// TwinCAT 3 PLC project Untitled1
// ProgramVersion: 3.1.4023.0
// libraries:
//   Tc2_ControllerToolbox, * (Beckhoff Automation GmbH)
//   Tc2_Standard, * (Beckhoff Automation GmbH)
//   Tc2_System, * (Beckhoff Automation GmbH)
//   Tc2_TempController, * (Beckhoff Automation GmbH)
//   Tc2_Utilities, * (Beckhoff Automation GmbH)
//   Tc3_EventLogger, * (Beckhoff Automation GmbH)
//   Tc3_Module, * (Beckhoff Automation GmbH)
// project tree:
//   DUTs/01_系统/ ST_AlarmID.TcDUT, ST_AlarmString.TcDUT, ST_Input.TcDUT, ST_Output.TcDUT, ST_Setting.TcDUT, ST_States.TcDUT
//   DUTs/Data types Alarm/ Alm_AlarmHistoryType.TcDUT, Alm_AlarmType.TcDUT, Alm_AlmMsg.TcDUT, Alm_EventClass.TcDUT
//   DUTs/ ST_Point.TcDUT
//   DUTs/文件配方/ FB_FileOperate.TcPOU
//   DUTs/文件配方/Swen_Products/ FB_DirectoryCopy.TcPOU, FB_FileCopy.TcPOU, FB_FileCopy_lib.TcPOU
//   GVLs/ Visu_Variables_HideInput.TcGVL, _01_Global_Variables.TcGVL, _04_Global_Variables_InOutput.TcGVL, _10_Global_Variables_Alarm.TcGVL, _12_Global_Variables_PeiFan.TcGVL
//   / PlcTask.TcTTO
//   POUs/ Controller_v2.TcPOU, FB_Actuator.TcPOU, Line_chart.TcPOU, MAIN.TcPOU
//   POUs/EventGridTest/ EventGrid.TcPOU
//   POUs/报警/ FB_AlarmMain.TcPOU, FB_SetAlarm.TcPOU, MAIN_Alarm.TcPOU, SW_FormatWstring.TcPOU
//   POUs/文件记录/ data_save.TcPOU, FB_DiagDataLogging.TcPOU
// real-time tasks:
//   TASK PlcTask: cycle T#10ms, priority 20, ADS port 350

CONFIGURATION Untitled1
    RESOURCE PLC ON TwinCAT3
        TASK PlcTask(INTERVAL := T#10ms, PRIORITY := 20);
        PROGRAM MAIN WITH PlcTask : MAIN;
    END_RESOURCE
END_CONFIGURATION

// ---- DUTs/01_系统/ST_AlarmID.TcDUT
TYPE ST_AlarmID :
(*报警的id号，swen*)
STRUCT
	(*系统*)
	EtherCATBusErr:					INT:=1;(*EtherCAT总线错误*)
	SystemLoading:					INT:=2;(*系统启动中*)
	EmergentStop:					INT:=3;(*急停按钮*)
	ProductChangeNeedSave:			INT:=4;
	ProductLoadingNoPowerOff:		INT:=5;
	AirPressLow:					INT:=6;(*气压低!*)
	Prushing:						INT:=7;(*暂停中*)
	NeedHoming:						INT:=8;(*开机前请先找原点*)
	IsHoming:						INT:=9;(*正在找原点*)
	AutoStoping:					INT:=10;(*自动停机中*)
	AutoStopImediery:				INT:=11;(*马上停机中*)
	AutoRuning:						INT:=12;(*设备运行中*)
	ComErrorVS:						INT:=13;(*视觉控制器通讯异常*)
	ServoError:						INT:=14;(*伺服出错*)
	ServoHwError:					INT:=15;(*伺服驱动器报错，硬件报错*)
	ServoLimit:						INT:=16;(*伺服驱动器限位到*)
	CycleTimeOut:					INT:=17;(*循环时间超时*)
	ModbusRtuError:					INT:=18;(*ModbusRtu总线错误*)
	RobotError1:					INT:=19;(*机器人错误*)
	RobotError2:					INT:=20;(*机器人错误*)
	StepServoError:					INT:=21;(*步进驱动器报错*)
	RobotSN_Error:					INT:=22;(*机器人序列号异常*)

	(*程序逻辑*)
	ClampVacuum:					INT:=26;(*机器人1真空吸取失败*)








	(*序列号*)
	Machime_SoftHwDif:				INT:=50;(*软硬件不匹配*)
	Machime_Alarm_NeedKey:			INT:=51;(*系统即将进入维护模式*)
	Machime_Stop_NeedKey:			INT:=52;(*系统已经进入维护模式*)

END_STRUCT
END_TYPE

// ---- DUTs/01_系统/ST_AlarmString.TcDUT
TYPE ST_AlarmString :
STRUCT
	chinese:		STRING:='CN';
	english:		STRING:='EN';
END_STRUCT
END_TYPE

// ---- DUTs/01_系统/ST_Input.TcDUT
TYPE ST_Input :
STRUCT
	biSnAirPressOk:				BOOL;(*压缩气源正常*)
	biSnBackDoorIsClose:				BOOL;(*后门关*)

	biSwEmgStop:				BOOL;(*急停按钮*)
	biBtStart:				BOOL;(*开始按钮*)
	biBtStop:				BOOL;(*停止按钮*)
	biBtHold:				BOOL;(*暂停按钮*)

   	biSnVacuuSor:				BOOL;(*取料真空检测*)

	biSnConvBoxIn:				BOOL;(*检测到进料口有箱子进来了*)
	biSnConvBoxOut:				BOOL;(*检测到出料口有箱子需要出来*)
	biSnBoxCapper:				BOOL;(*封箱机检测到有箱子进来*)


	noUse:				BOOL;





END_STRUCT
END_TYPE

// ---- DUTs/01_系统/ST_Output.TcDUT
TYPE ST_Output :
STRUCT


  	bqBoxCapperDw     (*	 压箱气缸	*)	,
  	bqBoxCapperCut      (*	剪断气缸  	*)	,

	bqClamperSuck	(*	机械手吸真空		*)	,
 	bqClamperZBrake          (*Z伺服刹车*)	,

	bqLightGrean(*绿灯 *)	,
 	bqLightYellow(*黄灯*)	,
 	bqLightRed(*红灯*)	,
 	bqBuzzer(*蜂鸣器*)	,

	noUse:				BOOL;

END_STRUCT
END_TYPE

// ---- DUTs/01_系统/ST_Setting.TcDUT
TYPE ST_Setting :
STRUCT
	(*系统*)
	gcSimulationMode:		BOOL;
	JogVelocity:			REAL:=20;
	AutoVelocity:			REAL:=500;(*皮带的速度*)
	ClampVelocity:			REAL:=2000;(*机械手的速度*)

	tCutTime:				REAL:=0.5;(*剪断时间*)

	ZPickUpHeight:			REAL:=200;(*抓起来的高度*)
	XPlacePos:				REAL:=450;(*抓过去的X距离*)
	YPlacePos:				REAL:=330;(*抓过去的Y距离*)
	ZPlacePos:				REAL:=-650;(*放到地板的高度*)
	Box_Longth:				REAL:=215;(*箱子长*)
	Box_Width:				REAL:=190;(*箱子宽*)
	Box_Height:				REAL:=198;(*箱子高*)

END_STRUCT
END_TYPE

// ---- DUTs/01_系统/ST_States.TcDUT
TYPE ST_States :
STRUCT
	ManualModeIsActive:				BOOL;(*手动模式*)
	AutoModeIsActive:				BOOL;(*自动模式*)
	MachineRunInCycle:				BOOL;(*自动运行中*)
	GoPauseState:					BOOL;(*请求暂停记忆*)
	AutoStoping:						BOOL;(*自动停机中*)
	ResetAlarm:						BOOL;(*报警复位*)
	GoHome:							BOOL;(*请求找原点*)


	(*电机*)
	HomeDone:						BOOL;(*原点完成*)
	Motor_PowerOn:				BOOL;(*上电完成*)
	Motor_HomeDone:				BOOL;(*原点完成*)
	Motor_SwError:				BOOL;(*电机NC软件出错*)
	Motor_SwErrId:				UDINT;
	Motor_Limit:				BOOL;(*电机限位*)
	Motor_HwError:				BOOL;(*电机硬件出错*)

	Hmi_btHome:						BOOL;(*画面按钮*)(*回原点*)
	Hmi_btAutoRun:					BOOL;(*画面按钮*)(*开始*)
	Hmi_btAutoStop:					BOOL;(*画面按钮*)(*停止*)
	Hmi_btPause:					BOOL;(*画面按钮*)(*暂停*)


	(*状态*)
	ConvCanRun:						BOOL:=TRUE;(*传送带启动允许*)

	ActBoxId:						INT;(*当前进箱子的ID号*)


END_STRUCT
END_TYPE

// ---- DUTs/Data types Alarm/Alm_AlarmHistoryType.TcDUT
TYPE Alm_AlarmHistoryType :
STRUCT
  	EventMessage:            	WSTRING;
	EventId:					INT;
   	EventTime:               	DT;
END_STRUCT
END_TYPE

// ---- DUTs/Data types Alarm/Alm_AlarmType.TcDUT
TYPE Alm_AlarmType :
STRUCT
      (*InPut*)
	EventId:					INT;
    EventMessage:			WSTRING;
    EventTime:                                 DT;
	EventActive:				BOOL;
	QuitRequired:				BOOL;
	QuitEvent:				BOOL;
	EventClass:				Alm_EventClass;
	AlarmMsg:				Alm_AlmMsg;
	AlarmlampOn:			BOOL;(*报警灯*)
	AutoRunOff:				BOOL;(*退出自动循环*)

	(* event actions OutPut	*)
	AlarmAction1:				BOOL;
	AlarmAction2:				BOOL;
	AlarmAction3:				BOOL;
	AlarmAction4:				BOOL;
	AlarmAction5:				BOOL;
	AlarmAction6:				BOOL;
	AlarmAction7:				BOOL;
	AlarmAction8:				BOOL;

       (*OutPut*)
	EventAlive:					BOOL;
    ShowlampOn:           		BOOL;
	InUse:                		BOOL;
END_STRUCT
END_TYPE;

// ---- DUTs/Data types Alarm/Alm_AlmMsg.TcDUT
TYPE Alm_AlmMsg :
STRUCT
	CN:		WSTRING:="中文";
	EN:		STRING:='En';	
END_STRUCT
END_TYPE

// ---- DUTs/Data types Alarm/Alm_EventClass.TcDUT
TYPE Alm_EventClass :
(
    NoAlarm                  :=0,(*无警报*)
    Message_1      :=1,(*信息*)
    Event_2            :=2,(*事件*)
    non_3                        :=3,(*暂无*)
    non_4                       :=4,(*暂无*)
    non_5                         :=5,(*暂无*)
    Alarm_6          :=6,(*不停机警报*)
    Stop_7                :=7(*停机警报*)
);
END_TYPE

// ---- DUTs/ST_Point.TcDUT
TYPE ST_Point :
STRUCT
	x : LREAL;
	y : LREAL;
END_STRUCT
END_TYPE

// ---- GVLs/Visu_Variables_HideInput.TcGVL
{attribute 'Tc2GvlVarNames'}
VAR_GLOBAL

	(*
		User Level Control
	*)
	sUserLevel:					STRING[20];
	nVisuUserLevel:				INT;
	bUseLogOutDelay:			BOOL;
	fUserLogOutDelay:			LREAL;
	sUserPassword:				STRING[20];
	bUserLevel0:				BOOL;
	bUserLevel1:				BOOL;
	bUserLevel2:				BOOL;
	bUserLevel3:				BOOL;
	bNewPassword:				BOOL;
	sNewUserPass1:			STRING[20];
	sNewUserPass2:			STRING[20];
	oldPasswords:				ARRAY [0..7] OF STRING[20];
	oldLanguage:				STRING[40];
	bVisuExUserLevel:			BOOL;
	bVisuInUserLevel:			BOOL;

(* ######################### Pswd Input Varaibles ########################## *)

	sPassInput : STRING := '';
	sPassV : STRING;

	i: DINT;
	iLen: DINT;
	bReset: BOOL;

	b_a_s : BOOL;
	b_b_s : BOOL;
	b_c_s : BOOL;
	b_d_s : BOOL;
	b_e_s : BOOL;
	b_f_s : BOOL;




	b_1_s : BOOL;
	b_2_s : BOOL;
	b_3_s : BOOL;
	b_4_s : BOOL;
	b_5_s : BOOL;
	b_6_s : BOOL;
	b_7_s : BOOL;
	b_8_s : BOOL;
	b_9_s : BOOL;
	b_0_s : BOOL;



	bBack: BOOL;
	iBackLen: INT;
	bShowNumPad:	BOOL;
	bHideNumPad:	BOOL;
	bCmdShowNumPad: BOOL;
	bCmdEnterValue:	BOOL;
	bCmdEscNumPad:	BOOL;
	sChangedPswd: STRING;

	bCmdShowNumPadUserPswd:	BOOL;
	bCmdShowNumPadNewPswd1:	BOOL;
	bCmdShowNumPadNewPswd2:	BOOL;

	sUserPasswordHide	:	STRING[20];
	sNewUserPass1Hide:	STRING[20];
	sNewUserPass2Hide:	STRING[20];

	bHidePswdFlush:	BOOL;

END_VAR

// ---- GVLs/_01_Global_Variables.TcGVL
{attribute 'Tc2GvlVarNames'}
VAR_GLOBAL
	DATA:						ST_States;	(*状态*)
//	gBox: 						ARRAY[0..23] OF ST_Box;(*箱子的状态*)
//	CLAMP:						APP_Clamp;(*实例化FB APP_Clmap*)
//	CONV:						APP_Conv;(*实例化FB APP_Conv*)

	RqSysManualModeIsActive,		(*需要在手动模式*)
	RqSysAutoModeIsActive,			(*需要在自动模式*)
	RqSysGoHome:				BOOL;(*需要回原点信号*)
	RqSysMachineRunInCycle: 	BOOL;(*需要设备在循环运行模式*)
	RqSysGoPauseState: 			BOOL;(*需要设备暂停*)
	Tem_Act			:LREAL;
	Tem_Act_1		:LREAL;
	Tem_control		:LREAL;
	Tem_control_1	:LREAL;
END_VAR
VAR_GLOBAL PERSISTENT(*断电保存型变量*)
	SET:							ST_Setting;	(*当前设定值*)
END_VAR

// ---- GVLs/_04_Global_Variables_InOutput.TcGVL
{attribute 'Tc2GvlVarNames'}
VAR_GLOBAL(*输入输出*)

	(*程序用变量*)
	stInput:				ST_Input;
	stOutput:				ST_Output;

	(*链接到硬件的变量*)
	EL1889 AT%I*: 			ARRAY[1..20,1..16] OF BOOL;
	EL2889 AT%Q*: 			ARRAY[1..20,1..16] OF BOOL;
END_VAR

// ---- GVLs/_10_Global_Variables_Alarm.TcGVL
{attribute 'Tc2GvlVarNames'}

VAR_GLOBAL(*报警库设置*)

	gbAlarm_NoStopAlarm,
	gbAlarm_StopAlarm ,
	gbAlarm_ShowlampOn ,
	gbAlarm_FalshLamp ,
	gbAlarm_NeedPause ,
	gbAlarm_ExtruderOff ,
	gbAlarm_HydraulicOff ,
	gbAlarm_HeatingOff ,
	gbAlarm_FillingOff ,
	gbAlarm_ServoMotorOff ,
	gbAlarm_AutoRunOff ,
	gbAlarm_AlarmAction1 ,
	gbAlarm_AlarmAction2 ,
	gbAlarm_AlarmAction3 ,
	gbAlarm_AlarmAction4 ,
	gbAlarm_AlarmAction5 ,
	gbAlarm_AlarmAction6 ,
	gbAlarm_AlarmAction7 ,
	gbAlarm_AlarmAction8	:	BOOL;

	gbHMIAlarmReset:		BOOL;
	AlarmID:				ST_AlarmID;
	//fbSetAlarm:				ARRAY[0..cnAlarmLast ] OF FB_SetAlarm;(*报警功能块数组*)
	HMI_AlarmActive:		ARRAY[cnAlarmFirst..cnAlarmLast ] OF BOOL;(*当前激活的报警数组*)(*给HMI用*)

END_VAR

VAR_GLOBAL
	  	Alm_ActiveAlarmNum:             	INT;(*当前激活警报的数量*)
	 	Alm_HistoryAlarmNum:           		INT;(*历史警报的数量*)
	 	AlarmActionArray:					ARRAY [cnAlarmFirst..cnAlarmLast] OF Alm_AlarmType;(*记录所有警报状态的数组*)
		AlarmActiveArray:					ARRAY [cnAlmActiveFirst..cnAlmActiveLast] OF Alm_AlarmHistoryType;(*记录已激活警报状态的数组*)
		fbSetAlarm:							ARRAY[cnAlarmFirst..cnAlarmLast] OF FB_SetAlarm;

	  	Alm_bHMIClearHistory:            	BOOL;(*清除历史报警*)
		Alm_bBtReset:						BOOL;//报警清除按钮
	  	Alm_iHMIAlarmID:                 	INT;(*当前报警id,给循环显示用*)
		tActSystemTime: 					TIMESTRUCT;//当前系统时间
		gwsActEventMsg:						WSTRING;//当前显示的报警信息，跑马灯形式
		gsWriteToLog:						STRING;//当前需要添加到报警历史文件的信息
		CurrentLanguage:					STRING;
END_VAR

VAR_GLOBAL PERSISTENT(*断电保存型变量,历史报警*)
	   	AlarmHistoryArray :				ARRAY [cnAlmHistoryFirst..cnAlmHistoryLast] OF Alm_AlarmHistoryType;(*记录历史警报状态的数组*)
END_VAR

(*
-------------------------------------在调用的程序里请定义如下变量:----------------------------------------------
*)
VAR_GLOBAL CONSTANT
		cnAlarmFirst:                             	INT:=1;(*报警的最小id号*)(*默认为1，不需改动*)
		cnAlarmLast:                             	INT:=50;(*报警的最大id号*)
		cnAlmActiveFirst:                       	INT:=1;(*当前激活的警报最小id号*)(*默认为1，不需改动*)
		cnAlmActiveLast:                       		INT:=20;(*当前激活的警报最大id号*)
		cnAlmHistoryFirst:                    		INT:=1;(*历史警报最小id号*)(*默认为1，不需改动*)
		cnAlmHistoryLast:                   	 	INT:=200;(*历史警报最大id号*)
END_VAR

// ---- GVLs/_12_Global_Variables_PeiFan.TcGVL
{attribute 'Tc2GvlVarNames'}
VAR_GLOBAL CONSTANT(*配方*)
	cnMaxRecepeNum:		INT:=25;
END_VAR
VAR_GLOBAL
	vbtRecipeArr:				ARRAY[1..cnMaxRecepeNum] OF BOOL;
	strRecipeArr:				ARRAY[1..cnMaxRecepeNum] OF STRING;
	vbtFlash:					BOOL;
	vbtLoad:					BOOL;
	vbtSave:					BOOL;
	vbtDel:						BOOL;
	vbtLoadFromUSB:				BOOL;
	vbtSaveToUSB:				BOOL;
	ShowDiag: 					BOOL;
	DiagIndex:					INT;
	iSelectIndex:				INT;//当前选择的id号
	vbtYes: 					BOOL;
	vbtNo: 						BOOL;
	strShowDiagName:			STRING;
END_VAR
VAR_GLOBAL PERSISTENT
	strInputReceipeName AT%Q*:		STRING(30);(*需要保存到NovRam*)
	strCurrentReceipeName AT%Q*:	STRING(30);(*需要保存到NovRam*)
END_VAR

// ---- POUs/MAIN.TcPOU
PROGRAM MAIN
VAR
	(* 选择功能块，温度控制库有两个功能块版本 V1和 V2 ，系统通过默认选择 V1，V1为旧版本，已被淘汰 *)
	nSelectController	: UINT := 1;	
	
(* 激活系统触发条件 *)	
	bStartTemControl	: BOOL;		
	timer1				:ton;
	ton1				:ton;
	ton2				:ton;
	light1				:BOOL;
	light2				:BOOL;
	Pt2					:TIME:=T#10D;
	Et2					:TIME;
	Tnowtotaltime		:REAL;
	clk1				:R_trig;
	act_1:FB_Actuator;
	enable,lockbyitself,manualmode,simumode:BOOL;
	s_rqwork,s_rqbasic:BOOL;
	sensor AT %I*:ARRAY[0..7] OF BOOL;//输入信号 DI1-DI8
	output AT %Q*:ARRAY[0..7] OF BOOL;//输出信号 DO1-DO8
END_VAR

(* 调用功能块V2，需将nSelectController从1切换为2 *)
	timer1(IN:=  bStartTemControl, PT:=Pt2 , Q=> , ET=>Et2 );
	clk1(CLK:=bStartTemControl , Q=> );
MAIN_ALarm();
EventGrid();	
IF 	bStartTemControl THEN
	
	nSelectController:= 2  ;   
	
	Line_chart();		
	data_save();
	Tem_Act:=Controller_v2.iTempre_Compare;
	Tem_Act_1:=Tem_Act/10;
	Tem_control:=Controller_v2.iTempre;
	Tem_control_1:=Tem_control/10;
END_IF;
	Tnowtotaltime:=TIME_TO_REAL(Et2)/1000;
	

	Controller_v2();
	
ton1(IN:=NOT ton2.Q, PT:=T#2000MS, Q=> light1, ET=> );
ton2(IN:= ton1.Q, PT:= T#2000MS, Q=> , ET=> );
IF NOT ton1.Q THEN
	light2:=TRUE;
	ELSE
	light2:=FALSE;	
	
END_IF
(*===================================================================*)
act_1(
	benable:= enable, 
	inWork:= sensor[0], 
	inBasic:= sensor[1], 
	FilterInWork:= T#20MS, 
	FilterInBasic:= T#20MS, 
	rqWork:= s_rqwork, 
	rqBasic:= s_rqbasic, 
	TimeOutWork:= , 
	TimeOutBasic:= , 
	bUseTimeLimit:= simumode, 
	bLockByItself:= lockbyitself, 
	bForceEnableManualBt:= manualmode, 
	sName:= "actor1", 
	doWork=> output[0], 
	doBasic=> output[1], 
);

END_PROGRAM

// ---- POUs/FB_Actuator.TcPOU
FUNCTION_BLOCK FB_Actuator(*执行器*)
VAR_INPUT
	benable:					BOOL;(*使能信号*)
	inWork:					BOOL;(*在工作位的信号输入*)
	inBasic:					BOOL;(*在基本位的信号输入*)
	FilterInWork:				TIME;(*在工作位滤波时间*)
	FilterInBasic:				TIME;(*在基本位滤波时间*)
	rqWork:					    BOOL;(*到工作位指令*)
	rqBasic:					BOOL;(*到基本位指令*)
	EnableManuWorkBt:		BOOL:=TRUE;(*使能到工作位按钮*)
	EnableManuBasicBt:		BOOL:=TRUE;(*使能到基本位按钮*)
	TimeOutWork:			REAL:=5;(*到工作位超时报警时间*)(*单位s*)
	TimeOutBasic:			REAL:=5;(*到基本位超时报警时间*)(*单位s*)
	bUseTimeLimit:			BOOL:=FALSE;(*利用时间做限位到位开关，不使用实际的反馈点*)
	bLockByItself:				BOOL;(*是否自锁*)
	bForceEnableManualBt:		BOOL;(*强制使用手动按钮功能,不需要转换到手动模式*)
	breset:BOOL;(*复位按钮*)
	sName:					WSTRING:="执行器";
END_VAR
VAR_OUTPUT
	isWork:					BOOL;(*已经到了工作位*)
	isBasic:				BOOL:=TRUE;(*已经到了基本位*)
	doWork:					BOOL;(*开始到工作位输出信号*)
	doBasic:				BOOL;(*开始到基本位输出信号*)
	bError:					BOOL;(*错误*)
	ierrorID:					INT;(*错误代码，参考action errorID*)
	MoveWorkTime:			REAL;(*到工作位时间计时*)(*单位s*)
	MoveBasicTime:			REAL;(*到基本位时间计时*)(*单位s*)
END_VAR
VAR
	btManuWork:				BOOL;(*手动按钮*)(*工作位*)
	btManuBasic:				BOOL;(*手动按钮*)(*基本位*)
	timecountwork:BOOL;(*工作位计时信号*)
	timecountbasic:BOOL;(*基本位计时信号*)
	R_TRIG_TIMECOUNT:		ARRAY[1..4] OF R_TRIG;
	timeCount:				ARRAY[1..2] OF TON;
	Filter:					ARRAY[1..2] OF TON;
	R_TRIG_TimeOut: 		ARRAY[1..2] OF R_TRIG;
END_VAR

//错误ID报警信息
(*
0：没有错误；
1：自动模式同时触发rqwork和rqbasic；
2：手动模式同时触发btmanuwork和btmanubasic；
3：未给manuworkbt按钮使能；
4：未给manubasicbt按钮使能；
5：工作位运行超时；
6：基本位运行超时；
*)
IF benable AND NOT berror THEN
(*==============安全，防止请求工作位和请求基本位逻辑同时触发造成事故=============================*)
IF rqWork
AND rqBasic THEN 
	rqWork:=rqBasic:=FALSE; 
	bError:=TRUE;
	ierrorID:=1;
END_IF
IF btManuWork 
AND btManuBasic THEN
	btManuWork:=btManuBasic:=FALSE; 
	bError:=TRUE;
	ierrorID:=2;
END_IF

(*==============自动模式的输出=============================*)
IF NOT bForceEnableManualBt //未触发强制使用手动
(*AND (RqSysAutoModeIsActive//系统请求自动模式
	OR DATA.GoHome) *)THEN
	IF bLockByItself THEN	(*触发了自锁模式，持续输出工作位/基本位信号*)
		IF rqWork THEN //请求到工作位
			doWork:=TRUE;//锁定工作位
			doBasic:=FALSE;
		ELSIF rqBasic THEN//请求到基本位
			doWork:=FALSE;
			doBasic:=TRUE;//锁定基本位
		END_IF
	ELSE					(*未触发自锁，进入普通模式，输出信号自动复位*)
		doWork:=rqWork
				(*OR (btManuWork
				AND DATA.ManualModeIsActive
				AND EnableManuWorkBt)*);
		doBasic:=rqBasic
				(*OR (btManuBasic
				AND DATA.ManualModeIsActive
				AND EnableManuBasicBt)*);
	END_IF

(*==============手动模式的输出=============================*)
ELSIF (*RqSysManualModeIsActive//系统请求使用手动模式
OR*) bForceEnableManualBt THEN//强制使用手动模式

	IF bLockByItself THEN	(*自锁模式*)
		IF btManuWork//使能并触发手动按钮请求工作位
		AND EnableManuWorkBt THEN
			doWork:=TRUE;//锁定工作位
			doBasic:=FALSE;
		ELSIF btManuBasic//使能并触发手动按钮请求基本位
		AND EnableManuBasicBt THEN
			doWork:=FALSE;
			doBasic:=TRUE;//锁定基本位
		END_IF
	ELSE					(*普通模式，信号自复位*)
		doWork:=btManuWork
				AND EnableManuWorkBt;//到工作位=手动按钮工作位 且 使能该按钮
		doBasic:=btManuBasic
				AND EnableManuBasicBt;//到基本位=手动按钮基本位 且 使能该按钮
	END_IF

ELSIF NOT bLockByItself THEN
	doWork:=FALSE;
	doBasic:=FALSE;
END_IF

(*=========================状态输出=============================*)
IF (*Set.gcSimulationMode(*程序模拟运行*)
OR *)bUseTimeLimit THEN(*利用时间做限位到位开关，不使用实际的反馈点*)
	IF doWork THEN
		Filter[1](IN:=doWork , PT:=T#1S , Q=>isWork);
		isBasic:=FALSE;
	ELSE
		Filter[1](IN:=FALSE);
	END_IF
	IF doBasic THEN
		Filter[2](IN:=doBasic , PT:=T#1S , Q=>isBasic);
		isWork:=FALSE;
	ELSE
		Filter[2](IN:=FALSE);
	END_IF

ELSE(*实际输入输出*)
	IF FilterInWork>T#0ms THEN
		Filter[1](IN:=inWork , PT:=FilterInWork , Q=>isWork);
	ELSE
		isWork:=inWork;
	END_IF
	IF FilterInWork>T#0ms THEN
		Filter[2](IN:=inBasic , PT:=FilterInBasic , Q=>isBasic);
	ELSE
		isBasic:=inBasic;
	END_IF
END_IF


(*==============手动时，条件不满足报警输出============================*)
IF (*DATA.ManualModeIsActive OR*) bForceEnableManualBt THEN
	IF btManuWork
	AND NOT EnableManuWorkBt THEN
		bError :=TRUE;
		ierrorID :=3;
	END_IF
	IF btManuBasic
	AND NOT EnableManuBasicBt THEN
		berror:=TRUE;
		ierrorID:=4;
	END_IF
END_IF


(*==============运动计时====================================================*)

R_TRIG_TIMECOUNT[1](CLK:= dowork, Q=> );
R_TRIG_TIMECOUNT[2](CLK:= iswork, Q=> );
R_TRIG_TIMECOUNT[3](CLK:= dobasic, Q=> );
R_TRIG_TIMECOUNT[4](CLK:= isbasic, Q=> );

IF r_trig_timecount[1].Q THEN
	timecountwork:=TRUE;
ELSIF r_trig_timecount[2].Q THEN
	MoveWorkTime:=0.002+TIME_TO_REAL(timeCount[1].ET)/1000;
ELSIF iswork THEN
	timecountwork:=FALSE;
END_IF

IF r_trig_timecount[3].Q THEN
	timecountbasic:=TRUE;
ELSIF r_trig_timecount[4].Q THEN
	MoveBasicTime:=0.002+TIME_TO_REAL(timeCount[2].ET)/1000;
elsif isbasic then
	timecountbasic:=FALSE;
END_IF

timeCount[1](IN:=timecountwork , PT:=T#1H );
timeCount[2](IN:=timecountbasic, PT:=T#1H );


(*==============报警====================================================*)
Act_Alarm();
END_IF

IF (*DATA.ResetAlarm OR*) breset THEN
	bError:=FALSE;
	ierrorID:=0;
	inWork:=FALSE;
	inBasic:=FALSE;
	rqWork:=FALSE;
	rqBasic:=FALSE;
END_IF

ACTION ACT_Alarm:
(*==============³¬Ê±±¨¾¯================================================================*)
R_TRIG_TimeOut[1](CLK:=TIME_TO_REAL(timeCount[1].ET)/1000 > TimeOutWork );
R_TRIG_TimeOut[2](CLK:=TIME_TO_REAL(timeCount[2].ET)/1000 > TimeOutBasic );

IF R_TRIG_TimeOut[1].Q THEN
	bError :=TRUE;
	ierrorID :=5;
END_IF

IF R_TRIG_TimeOut[1].Q THEN
	bError :=TRUE;
	ierrorID :=6;
END_IF
END_ACTION

END_FUNCTION_BLOCK

// ---- POUs/报警/MAIN_Alarm.TcPOU
PROGRAM MAIN_ALarm
VAR
	fbAlarmMAIN:				FB_AlarmMAIN;
	fbDiagDataLogging_S:		FB_DiagDataLogging;
	bInidDone: 					BOOL;
	D1:							DINT:=1;
	D2:							DINT:=1;
	ModleName:					STRING:='EL1008';
	TON_Delay:					TON;
	TON_TimeOutCount: 			TON;
END_VAR



IF NOT bInidDone THEN
	aInit();
ELSE
	TON_Delay(IN:=TRUE , PT:=T#2S );
	IF TON_Delay.Q THEN
		aOtherAlarm();
		fbAlarmMAIN();
		gbAlarm_StopAlarm := fbAlarmMAIN.AlarmAction1;
		gbAlarm_NeedPause := fbAlarmMAIN.AlarmAction2;
		fbDiagDataLogging_s(sInputString:=gsWriteToLog);
	END_IF		
END_IF

ACTION aInit:

	
	AlarmActionArray[1].AlarmMsg.CN	:=	"EtherCAT总线错误,模块名:%S";
	AlarmActionArray[2].AlarmMsg.CN	:=	"系统初始化中......";
	AlarmActionArray[3].AlarmMsg.CN	:=	"急停按钮!";
	AlarmActionArray[4].AlarmMsg.CN	:=	"配方参数改变，请注意保存配方!";
	AlarmActionArray[5].AlarmMsg.CN	:=	"配方系统运行中，请不要断开电源!";
	AlarmActionArray[6].AlarmMsg.CN	:=	"气压低!";
	AlarmActionArray[7].AlarmMsg.CN	:=	"暂停中!";
	AlarmActionArray[8].AlarmMsg.CN	:=	"开机前请先回原点";
	AlarmActionArray[9].AlarmMsg.CN	:=	"伺服正在找原点!";
	AlarmActionArray[10].AlarmMsg.CN	:=	"自动停机中!";
	AlarmActionArray[11].AlarmMsg.CN	:=	"立刻停机中!";
	AlarmActionArray[12].AlarmMsg.CN	:=	"设备自动运行中";
	AlarmActionArray[13].AlarmMsg.CN	:=	"视觉控制器通讯异常!";
	AlarmActionArray[14].AlarmMsg.CN	:=	"伺服NC报警,报警号:%S";
	AlarmActionArray[15].AlarmMsg.CN	:=	"伺服驱动器报错";
	AlarmActionArray[16].AlarmMsg.CN	:=	"伺服驱动器限位";
	AlarmActionArray[17].AlarmMsg.CN	:=	"系统时间超时!";
	AlarmActionArray[18].AlarmMsg.CN	:=	"ModbusRTU步进电机通讯异常!";
	AlarmActionArray[19].AlarmMsg.CN	:=	"机器人1信息提示!";
	AlarmActionArray[20].AlarmMsg.CN	:=	"机器人2信息提示!";
	AlarmActionArray[21].AlarmMsg.CN	:=	"步进驱动器报错!";
	AlarmActionArray[22].AlarmMsg.CN	:=	"机器人序列号异常!";

	
	AlarmActionArray[1].AlarmMsg.EN	:=	'EtherCATBusErr,At %S';
	AlarmActionArray[2].AlarmMsg.EN	:=	'SystemLoading';
	AlarmActionArray[3].AlarmMsg.EN	:=	'EmergentStop';
	AlarmActionArray[4].AlarmMsg.EN	:=	'ProductChangeNeedSave';
	AlarmActionArray[5].AlarmMsg.EN	:=	'ProductLoadingNoPowerOff';
	AlarmActionArray[6].AlarmMsg.EN	:=	'AirPressLow';
	AlarmActionArray[7].AlarmMsg.EN	:=	'Prushing';
	AlarmActionArray[8].AlarmMsg.EN	:=	'NeedHoming';
	AlarmActionArray[9].AlarmMsg.EN	:=	'IsHoming';
	AlarmActionArray[10].AlarmMsg.EN	:=	'AutoStoping';
	AlarmActionArray[11].AlarmMsg.EN	:=	'AutoStopImediery';
	AlarmActionArray[12].AlarmMsg.EN	:=	'AutoRuning';
	AlarmActionArray[13].AlarmMsg.EN	:=	'ComErrorVS';
	AlarmActionArray[14].AlarmMsg.EN	:=	'ServoError,ErrorId: %S';
	AlarmActionArray[15].AlarmMsg.EN	:=	'ServoHwError';
	AlarmActionArray[16].AlarmMsg.EN	:=	'ServoLimit';
	AlarmActionArray[17].AlarmMsg.EN	:=	'CycleTimeOut';
	AlarmActionArray[18].AlarmMsg.EN	:=	'ModbusRtuError';
	AlarmActionArray[19].AlarmMsg.EN	:=	'RobotError1';
	AlarmActionArray[20].AlarmMsg.EN	:=	'RobotError2';
	AlarmActionArray[21].AlarmMsg.EN	:=	'StepServoError';
	AlarmActionArray[22].AlarmMsg.EN	:=	'RobotSN_Error';
	
	
	FOR i:=cnAlarmFirst TO cnAlarmLast DO
		fbSetAlarm[i].EventId :=DINT_TO_INT( i);
	END_FOR	
	bInidDone:=TRUE;
END_ACTION

ACTION aOtherAlarm:

		fbSetAlarm[AlarmID.AirPressLow]
			(
			InUse:=			TRUE ,
			EventActive:=	NOT stInput.biSnAirPressOk ,
			FilterInUse:= 	TRUE,
			FilterTime:= 	T#20ms,
			QuitRequired:=	TRUE,
			QuitEvent:=		DATA.ResetAlarm ,
			EventClass:=	7 ,
			ToTheHistory:=	TRUE ,
			ToTheLogFile:=	TRUE,
			AlarmlampOn:=	TRUE ,
			(*急停*)AlarmAction1:=TRUE ,
			 );


		fbSetAlarm[AlarmID.EmergentStop]
			(
			InUse:=			FALSE ,
			EventActive:=	NOT stInput.biSwEmgStop ,
			FilterInUse:= 	TRUE,
			FilterTime:= 	T#20ms,
			QuitRequired:=	TRUE,
			QuitEvent:=		DATA.ResetAlarm ,
			EventClass:=	7 ,
			ToTheHistory:=	TRUE ,
			ToTheLogFile:=	TRUE,
			AlarmlampOn:=	TRUE ,
			(*急停*)AlarmAction1:=TRUE ,
			 );


		(*TON_TimeOutCount
			(
			IN:= 	MODE=AutoRuning
					AND ncAxis[1].Status.NotMoving
					AND ncAxis[2].Status.NotMoving
					AND ncAxis[3].Status.NotMoving
					AND ncAxis[4].Status.NotMoving
					AND ncAxis[5].Status.NotMoving
					AND ncAxis[6].Status.NotMoving
					AND ncAxis[7].Status.NotMoving
					AND ncAxis[8].Status.NotMoving
					AND ncAxis[9].Status.NotMoving
					AND ncAxis[10].Status.NotMoving,

			PT:=	T#5s
			);*);
		fbSetAlarm[AlarmID.CycleTimeOut]
			(
			InUse:=			FALSE,
			EventActive:=	TON_TimeOutCount.Q ,
			FilterInUse:= 	FALSE,
			FilterTime:= 	T#20ms,
			QuitRequired:=	TRUE,
			QuitEvent:=		DATA.ResetAlarm ,
			EventClass:=	7 ,
			ToTheHistory:=	TRUE ,
			ToTheLogFile:=	TRUE,
			AlarmlampOn:=	TRUE ,
			(*急停*)AlarmAction1:=TRUE ,
			 );

		fbSetAlarm[AlarmID.ServoError]
			(
			InUse:=			TRUE,
			EventActive:=	DATA.Motor_SwError ,
			FilterInUse:= 	FALSE,
			FilterTime:= 	T#20ms,
			QuitRequired:=	TRUE,
			QuitEvent:=		DATA.ResetAlarm ,
			EventClass:=	7 ,
			ToTheHistory:=	TRUE ,
			ToTheLogFile:=	TRUE,
			AlarmlampOn:=	TRUE ,
			(*急停*)AlarmAction1:=TRUE ,
			S1:=			UDINT_TO_STRING(DATA.Motor_SwErrId),
			 );
		DATA.Motor_SwError:=FALSE;

		fbSetAlarm[AlarmID.ServoHwError]
			(
			InUse:=			TRUE,
			EventActive:=	DATA.Motor_HwError ,
			FilterInUse:= 	FALSE,
			FilterTime:= 	T#20ms,
			QuitRequired:=	TRUE,
			QuitEvent:=		DATA.ResetAlarm ,
			EventClass:=	7 ,
			ToTheHistory:=	TRUE ,
			ToTheLogFile:=	TRUE,
			AlarmlampOn:=	TRUE ,
			(*急停*)AlarmAction1:=TRUE ,
			 );
		DATA.Motor_HwError:=FALSE;


		fbSetAlarm[AlarmID.ServoLimit]
			(
			InUse:=			TRUE,
			EventActive:=	DATA.Motor_Limit ,
			FilterInUse:= 	FALSE,
			FilterTime:= 	T#20ms,
			QuitRequired:=	TRUE,
			QuitEvent:=		DATA.ResetAlarm ,
			EventClass:=	3 ,
			ToTheHistory:=	TRUE ,
			ToTheLogFile:=	TRUE,
			AlarmlampOn:=	TRUE ,
			(*急停*)AlarmAction1:=FALSE ,
			 );
		DATA.Motor_Limit:=FALSE;



		fbSetAlarm[AlarmID.NeedHoming]
			(
			InUse:=			FALSE,
			EventActive:=	(DATA.Hmi_btAutoRun )
							AND NOT DATA.HomeDone ,
			FilterInUse:= 	FALSE,
			FilterTime:= 	T#20ms,
			QuitRequired:=	TRUE,
			QuitEvent:=		DATA.ResetAlarm ,
			EventClass:=	2 ,
			ToTheHistory:=	FALSE ,
			ToTheLogFile:=	FALSE,
			AlarmlampOn:=	FALSE ,
			 );

		fbSetAlarm[AlarmID.IsHoming]
			(
			InUse:=			TRUE,
			EventActive:=	RqSysGoHome ,
			FilterInUse:= 	FALSE,
			FilterTime:= 	T#20ms,
			QuitRequired:=	FALSE,
			QuitEvent:=		DATA.ResetAlarm ,
			EventClass:=	2 ,
			ToTheHistory:=	FALSE ,
			ToTheLogFile:=	FALSE,
			AlarmlampOn:=	FALSE ,
			 );

		fbSetAlarm[AlarmID.Prushing]
			(
			InUse:=			TRUE,
			EventActive:=	DATA.GoPauseState,
			FilterInUse:= 	FALSE,
			FilterTime:= 	T#20ms,
			QuitRequired:=	FALSE,
			QuitEvent:=		DATA.ResetAlarm ,
			EventClass:=	2 ,
			ToTheHistory:=	FALSE ,
			ToTheLogFile:=	FALSE,
			AlarmlampOn:=	FALSE ,
			AlarmAction2:=	TRUE,(*暂停*)
			 );

		fbSetAlarm[AlarmID.AutoRuning]
			(
			InUse:=			TRUE,
			EventActive:=	RqSysAutoModeIsActive
							AND NOT fbAlarmMain.ShowlampOn
							AND NOT DATA.GoPauseState
							AND NOT DATA.AutoStoping,
			FilterInUse:= 	FALSE,
			FilterTime:= 	T#20ms,
			QuitRequired:=	FALSE,
			QuitEvent:=		DATA.ResetAlarm ,
			EventClass:=	2 ,
			ToTheHistory:=	FALSE ,
			ToTheLogFile:=	FALSE,
			AlarmlampOn:=	FALSE ,
			 );

		fbSetAlarm[AlarmID.AutoStoping]
			(
			InUse:=			TRUE,
			EventActive:=	DATA.AutoStoping,
			FilterInUse:= 	FALSE,
			FilterTime:= 	T#20ms,
			QuitRequired:=	FALSE,
			QuitEvent:=		DATA.ResetAlarm ,
			EventClass:=	2 ,
			ToTheHistory:=	FALSE ,
			ToTheLogFile:=	FALSE,
			AlarmlampOn:=	FALSE ,
			 );
END_ACTION

END_PROGRAM

// ---- POUs/报警/FB_AlarmMain.TcPOU
FUNCTION_BLOCK FB_AlarmMAIN(*报警主程序,请调用一次*)
(*===========================================
by Swen 陈颂文
GuangZhou
2009-08-26
===========================================*)

VAR_INPUT
END_VAR
VAR_OUTPUT
	EventId:						INT;(*报警号.有报警时会轮询输出有报警的id号*)
   	EventMessage:                  	WSTRING;(*报警信息.有报警时会轮询输出有报警的id信息*)
	EventAlive:						BOOL;(*当前有报警*)
	EventClass:						Alm_EventClass;(*当前的最大报警等级*)
  	NoStopAlarm:                  	BOOL;(*有小于7的报警,不停机报警*)
   	StopAlarm:                     	BOOL;(*有大于6的报警,停机报警*)
   	ShowlampOn:                    	BOOL;(*报警灯亮*)
   	FalshLamp:                   	BOOL;(*报警灯闪亮.有报警时该信号闪烁输出*)

	AutoRunOff:					BOOL;(*退出自动循环*)
	AlarmAction1:				BOOL;(*用户定义报警动作*)(*例如定义为黄灯亮,则有报警号有触发时,该输出信号为1*)
	AlarmAction2:				BOOL;(*用户定义报警动作*)
	AlarmAction3:				BOOL;(*用户定义报警动作*)
	AlarmAction4:				BOOL;(*用户定义报警动作*)
	AlarmAction5:				BOOL;(*用户定义报警动作*)
	AlarmAction6:				BOOL;(*用户定义报警动作*)
	AlarmAction7:				BOOL;(*用户定义报警动作*)
	AlarmAction8:				BOOL;(*用户定义报警动作*)
END_VAR
VAR
	nConut:                                				INT;
   	fbFreePluse:                        				TON;
	m:                                          		INT;
	Resul:                                   			INT;
	n:                                            		INT;
	R_TRIG_AlarmShow:        							R_TRIG;
	R_TRIG_AlarmAlive:          						R_TRIG;
	FB_FreePluse_AlarmShow: 							TON;
	FB_FreePluse_AlarmAlive: 							TON;
	F_TRIG_bHMIClearHistory: 							F_TRIG;
	F_TRIG_EventAlive: 									F_TRIG;
	InstLocalSystemTime:								FB_LocalSystemTime;
END_VAR

(*Set Signal*)
 	EventAlive:=ShowlampOn:=AlarmAction1:=AlarmAction2:=AlarmAction3:=FALSE;
  	AlarmAction4:=AlarmAction5:=AlarmAction6:=AlarmAction7:=AlarmAction8:=FALSE;
	AutoRunOff :=	FALSE;(*退出自动循环*)
   	EventClass :=	0;

FOR nConut :=cnAlarmFirst TO cnAlarmLast DO
	    EventAlive :=	EventAlive OR AlarmActionArray[nConut].EventAlive;
	    ShowlampOn:=	ShowlampOn OR AlarmActionArray[nConut].ShowlampOn;
	    AlarmAction1:=	AlarmAction1 OR AlarmActionArray[nConut].AlarmAction1;
	    AlarmAction2:=	AlarmAction2 OR AlarmActionArray[nConut].AlarmAction2;
	    AlarmAction3:=	AlarmAction3 OR AlarmActionArray[nConut].AlarmAction3;
	    AlarmAction4:=	AlarmAction4 OR AlarmActionArray[nConut].AlarmAction4;
	    AlarmAction5:=	AlarmAction5 OR AlarmActionArray[nConut].AlarmAction5;
	    AlarmAction6:=	AlarmAction6 OR AlarmActionArray[nConut].AlarmAction6;
	    AlarmAction7:=	AlarmAction7 OR AlarmActionArray[nConut].AlarmAction7;
	    AlarmAction8:=	AlarmAction8 OR AlarmActionArray[nConut].AlarmAction8;
	    AutoRunOff :=	AutoRunOff 	OR AlarmActionArray[nConut].AutoRunOff;
	    EventClass  :=	MAX(EventClass,AlarmActionArray[nConut].EventClass);
END_FOR

(*Flash lamp*)
R_TRIG_AlarmShow(CLK:=ShowlampOn  );
IF ShowlampOn THEN
	IF R_TRIG_AlarmShow.Q THEN
		fbFreePluse(IN:=FALSE);
		FalshLamp:=TRUE;
	END_IF
	fbFreePluse(IN:=NOT fbFreePluse.Q,PT:=T#1S);
	IF fbFreePluse.Q THEN
		FalshLamp:=NOT FalshLamp;
	END_IF
ELSE
	FalshLamp:=FALSE;
END_IF


(*Action*)
AlarmAlive();
AlarmHMI();
AlarmShow();

(*Set Action*)
IF EventAlive THEN
     IF EventClass>6 THEN
         StopAlarm:=TRUE;
         NoStopAlarm:=FALSE;
     ELSE
         StopAlarm:=FALSE;
         NoStopAlarm:=TRUE;
    END_IF
ELSE
    StopAlarm:=FALSE;
    NoStopAlarm:=FALSE;
    EventId:=0;
    EventMessage:="";
    Alm_iHMIAlarmID:=0;
END_IF

	//获取系统时间
	InstLocalSystemTime(
		sNetID		:= '',
		bEnable		:= TRUE,
		dwCycle		:= 1,
		systemTime	=> tActSystemTime,
		);

ACTION AlarmAlive:

(*-----------------------------------当前报警列表显示-----------------------------*)
R_TRIG_AlarmAlive(CLK:=EventAlive);
IF EventAlive THEN
	IF R_TRIG_AlarmAlive.Q THEN
   	 	FB_FreePluse_AlarmAlive(In:=FALSE);
	END_IF
    FB_FreePluse_AlarmAlive(In:= NOT FB_FreePluse_AlarmAlive.Q,PT:=T#1S );
    IF FB_FreePluse_AlarmAlive.Q
	OR R_TRIG_AlarmAlive.Q THEN
         n:=cnAlarmFirst;
         m:=cnAlmActiveFirst;
          FOR n:=cnAlarmFirst TO cnAlarmLast DO
               IF AlarmActionArray[n].EventAlive THEN
                    AlarmActiveArray[m].EventId                  :=AlarmActionArray[n].EventId;
                   	AlarmActiveArray[m].EventMessage    :=		AlarmActionArray[n].EventMessage;						
                    AlarmActiveArray[m].EventTime            :=AlarmActionArray[n].EventTime;
                  	m:=m+1;
                    IF m>cnAlmActiveLast THEN
                       n:=32766;  (*exit FOR*)
                    END_IF
               END_IF
         END_FOR
         IF m<cnAlmActiveLast THEN
               FOR n:=m TO cnAlmActiveLast DO
                   AlarmActiveArray[n].EventId:=0;
                 	AlarmActiveArray[n].EventMessage:="";
                   	AlarmActiveArray[n].EventTime:=DT#2000-01-01-00:00;
             END_FOR
          END_IF
    END_IF
END_IF

F_TRIG_EventAlive(CLK:=EventAlive );
IF F_TRIG_EventAlive.Q THEN
	FOR n:=cnAlmActiveFirst TO cnAlmActiveLast DO 
		AlarmActiveArray[n].EventId:=0;
		AlarmActiveArray[n].EventMessage:="";
		AlarmActiveArray[n].EventTime:=DT#2016-01-01-00:00;
	END_FOR
END_IF
END_ACTION

ACTION AlarmHMI:


(*``````````````````````````````````````````清除历史报警`````````````````````````````````````*)
F_TRIG_bHMIClearHistory(CLK:=Alm_bHMIClearHistory  );
IF F_TRIG_bHMIClearHistory.Q THEN
       FOR n:=cnAlmHistoryFirst TO cnAlmHistoryLast DO
             AlarmHistoryArray[n].EventId:=0;
             AlarmHistoryArray[n].EventMessage:="";
             AlarmHistoryArray[n].EventTime:=DT#2016-01-01-00:00;
        END_FOR
        Alm_HistoryAlarmNum:=0;
END_IF
END_ACTION

ACTION AlarmShow:

(*-------------------------------跑马灯显示报警---------------------------------*)
FB_FreePluse_AlarmShow(IN:=NOT FB_FreePluse_AlarmShow.Q,PT:=T#1S );
IF FB_FreePluse_AlarmShow.Q 
OR R_TRIG_AlarmAlive.Q THEN
      n:=EventId;
      	FOR m:=n+1 TO cnAlarmLast DO
            IF AlarmActionArray[m].EventAlive THEN
                   n:=m;
                   m:=cnAlarmLast+10;
             END_IF;
      	END_FOR;
    	IF n<>EventId THEN
        	Resul:=n;     
   		ELSE
          	FOR m:=cnAlarmFirst TO cnAlarmLast DO
             	IF AlarmActionArray[m].EventAlive THEN
                 	n:=m;
                 	m:=cnAlarmLast+10;
              	END_IF;
          	END_FOR;
          	Resul:=n;
      	END_IF
END_IF

Alm_iHMIAlarmID:=EventId:=Resul;
IF EventId<=cnAlarmLast
AND EventId>= cnAlarmFirst THEN
	gwsActEventMsg:=EventMessage:=AlarmActionArray[EventId].EventMessage;
ELSE
	gwsActEventMsg:=EventMessage:="";	
END_IF
END_ACTION

END_FUNCTION_BLOCK

// ---- POUs/文件记录/FB_DiagDataLogging.TcPOU
FUNCTION_BLOCK FB_DiagDataLogging
(*==================================================================
历史文件夹操作
By SwenChen
at 20170809
===================================================================*)
VAR_INPUT
	bInUse:							BOOL:=TRUE;(*是否使能功能*)
	bCopyToUSB:						BOOL;(*把文件夹复制到u盘*)

	b_DiagDataLog_AutoDelete:		BOOL:=TRUE;	(* Auto Deletion of Logged Files / highly recommended!	*)(*是否自动删除文件*)
	n_DiagDataLog_KeepForWeeks:		INT:=4;

	bDiagDataLogRunOn_WinCE:		BOOL:=FALSE;
	cnst_DiagDataLogFilePath_XP:	STRING(255):='D:\';
	cnst_DiagDataLogFilePath_CE:	STRING(255):='Hard Disk\';

	cnst_USB_FilePath_XP:			STRING(255):='E:\';
	cnst_USB_FilePath_CE:			STRING(255):='Hard Disk2\';

	cnst_SubDir_DiagDataLog:		STRING(255):='DiagDataLog\';
	cnst_FileName:					STRING(255):='Sym';(*文件的前缀名*)

END_VAR
VAR_IN_OUT
	sInputString:					STRING;(*TC2只能是英文字符串，不能中文*)
END_VAR
VAR_OUTPUT
	bBusyWriting:					BOOL;
	sWriteData:						STRING;
END_VAR
VAR
	nTaskIdx:						BYTE:=0;
	fbGetTaskIdx:					GETCURTASKINDEX;
	fCycleTime:						LREAL;

	StartUp:						BOOL:=TRUE;
	count:							INT;
	dtemp:							DINT;
	dtemp2:							DINT;
	stemp:							STRING;
	btemp:							BOOL;

	aStringBuffer:					ARRAY[1..10] OF STRING;
	sActUseingString:				STRING;
	bInputDoWrite:					BOOL;

	nWrState:						INT;
	sWrite:							STRING(255);
	stWrTime:						TIMESTRUCT;
	fbFormat:						FB_FormatString;
	fbOpen:							FB_FileOpen;
	fbWrite:						FB_FileWrite;
	fbClose:						FB_FileClose;

	nState:							INT;
	nEntries:						INT;
	fbMakeDir:						FB_CreateDir;
	fbGetTime:						NT_GetTime;
	msecond:						UDINT;

	delstep:						INT:=0;
	CopyStep: 						INT:=0;
	deldatestart:					TIMESTRUCT;
	deldate:						TIMESTRUCT;
	fbdelete:						FB_FileDelete;
	fbDirectoryCopy:				FB_DirectoryCopy;
	fdeltime:						LREAL;
	ntemp:							INT;
	sFile:							STRING(255);
	bClearLined:					BOOL;

	bInitialWrite:					BOOL:=TRUE;
	bFirstLog:						BOOL:=TRUE;

	bDiagDataLog_Release : 			BOOL;
	stDiagDataLogTime:				TIMESTRUCT;

END_VAR

IF NOT bInUse THEN(*是否使能功能*)
	StartUp:=TRUE;
	RETURN;
END_IF

IF StartUp THEN
	(* get cycle time of this task	*)
	fbGetTaskIdx();
	nTaskIdx:=MAX(MIN(fbGetTaskIdx.index,4),1);
	fCycleTime:=UDINT_TO_LREAL(_TaskInfo[nTaskIdx].CycleTime)/10000000.0;
	nState:=0;
	IF fCycleTime<>0 THEN
		StartUp:=FALSE;
	END_IF
END_IF


act_CheckCom();		(*命令处理*)
act_AutoWrite();	(*写*)
act_AutoDelete();	(*删除旧文件*)
act_Copy2USB();		(*复制到其它文件夹*)

ACTION act_AutoDelete:

(*É¾³ý¾ÉÎÄ¼þ*)

CASE delstep OF
0:
	fdeltime:=10.0;
	IF b_DiagDataLog_AutoDelete AND (stDiagDataLogTime.wYear>0) AND (n_DiagDataLog_KeepForWeeks>0) THEN
		ntemp:=1+7*MIN(MAX(n_DiagDataLog_KeepForWeeks,4),4000);
		deldate:=stDiagDataLogTime;
		WHILE (ntemp>0) DO
			IF (deldate.wDay<2) THEN
				deldate.wDay:=deldate.wDay+28;
				deldate.wMonth:=deldate.wMonth-1;
				IF (deldate.wMonth<1) THEN
					deldate.wMonth:=12;
					deldate.wYear:=deldate.wYear-1;
				END_IF
			END_IF
			IF (deldate.wDay=ntemp) THEN
				deldate.wDay:=1;
				ntemp:=1;
			ELSIF (deldate.wDay>ntemp) THEN
				deldate.wDay:=deldate.wDay-ntemp;
				ntemp:=0;
			ELSE
				ntemp:=ntemp-deldate.wDay;
				deldate.wDay:=1;
			END_IF
		END_WHILE
		deldatestart:=deldate;
		delstep:=1;
	END_IF

1:	fdeltime:=fdeltime-fCycleTime;
	IF NOT b_DiagDataLog_AutoDelete THEN
		delstep:=0;
	ELSIF (fdeltime<=0.0) THEN
		delstep:=2;
	END_IF

2:
	IF bDiagDataLogRunOn_WinCE THEN
		sFile:=CONCAT(cnst_DiagDataLogFilePath_CE,cnst_SubDir_DiagDataLog);
	ELSE
		sFile:=CONCAT(cnst_DiagDataLogFilePath_XP,cnst_SubDir_DiagDataLog);
	END_IF
	sFile:=CONCAT(sFile,cnst_FileName);
	stemp:=WORD_TO_STRING(deldate.wYear);
	stemp:=CONCAT(stemp,'_');
	IF (deldate.wMonth<10) THEN
		stemp:=CONCAT(stemp,'0');
	END_IF
	stemp:=CONCAT(stemp,WORD_TO_STRING(deldate.wMonth));
	stemp:=CONCAT(stemp,'_');
	IF (deldate.wDay<10) THEN
		stemp:=CONCAT(stemp,'0');
	END_IF
	stemp:=CONCAT(stemp,WORD_TO_STRING(deldate.wDay));
	stemp:=CONCAT(stemp,'_');
	IF(deldate.wHour<10)THEN
		stemp:=CONCAT(stemp,'0');
	END_IF
	stemp:=CONCAT(stemp,WORD_TO_STRING(deldate.wHour));
	stemp:=CONCAT(stemp,'.LOG');
	fbdelete.sPathName:=CONCAT(sFile,stemp);
	fbdelete.bExecute:=TRUE;
	delstep:=3;

3:
	IF NOT fbdelete.bBusy THEN
		fbdelete.bExecute:=FALSE;
		IF (deldate.wHour=0) THEN
			deldate.wHour:=23;
			deldate.wDay:=deldate.wDay-1;
		ELSE
			deldate.wHour:=deldate.wHour-1;
		END_IF
		IF (deldate.wDay<1) THEN
			deldate.wDay:=31;
			deldate.wMonth:=deldate.wMonth-1;
		END_IF
		IF (deldate.wMonth<1) THEN
			deldate.wMonth:=12;
			deldate.wYear:=deldate.wYear-1;
		END_IF
		fdeltime:=1.5;
		dtemp2:=12*WORD_TO_DINT(deldatestart.wYear-deldate.wYear)+WORD_TO_DINT(deldatestart.wMonth-deldate.wMonth);
		IF (dtemp>24) THEN
			delstep:=0;
		ELSE
			delstep:=1;
		END_IF
	END_IF

ELSE
	delstep:=0;

END_CASE

fbdelete();
END_ACTION

ACTION act_AutoWrite:

(*Ð´*)

CASE nState OF

0:	(*
		wait for clearance
	*)
	nEntries:=0;
	bInputDoWrite:=bDiagDataLog_Release:=FALSE;
	nWrState:=0;
	IF NOT StartUp THEN
		nState:=1;
	END_IF

1:	(*
		try to create the directory
	*)
	fbMakeDir.bExecute:=FALSE;
	fbGetTime.START:=FALSE;
	fbMakeDir.sNetId:='';
	IF bDiagDataLogRunOn_WinCE THEN
		fbMakeDir.sPathName:=CONCAT(cnst_DiagDataLogFilePath_CE,cnst_SubDir_DiagDataLog);
	ELSE
		fbMakeDir.sPathName:=CONCAT(cnst_DiagDataLogFilePath_XP,cnst_SubDir_DiagDataLog);
	END_IF
	fbMakeDir.ePath:=PATH_GENERIC;
	fbMakeDir.tTimeout:=T#5s;
	nState:=2;

2:	fbMakeDir();
	fbGetTime();
	IF NOT fbMakeDir.bExecute THEN
		fbMakeDir.bExecute:=TRUE;
	ELSIF NOT fbMakeDir.bBusy THEN
		IF NOT fbGetTime.START THEN
			fbGetTime.START:=TRUE;
		ELSIF NOT fbGetTime.BUSY THEN
			IF fbGetTime.ERR THEN
				stDiagDataLogTime.wYear:=stDiagDataLogTime.wMonth:=stDiagDataLogTime.wDay:=0;
				stDiagDataLogTime.wHour:=stDiagDataLogTime.wMinute:=stDiagDataLogTime.wSecond:=0;
				stDiagDataLogTime.wMilliseconds:=0;
				msecond:=0;
			ELSE
				stDiagDataLogTime:=fbGetTime.TIMESTR;
				msecond:=fbGetTime.TIMESTR.wMilliseconds;
			END_IF
			fbGetTime(START:=FALSE);
			fbMakeDir(bExecute:=FALSE);
			nState:=11;
		END_IF
	END_IF


11:
	IF(nState>=10)THEN
		(*
			update and/or synchronize the clock
		*)
		stDiagDataLogTime.wMilliseconds:=stDiagDataLogTime.wMilliseconds+LREAL_TO_WORD(MIN(MAX(1000.0*fCycleTime,1.0),30000.0));
	
		IF(stDiagDataLogTime.wMilliseconds>=1000)THEN
			stDiagDataLogTime.wMilliseconds:=stDiagDataLogTime.wMilliseconds-1000;
			stDiagDataLogTime.wSecond:=stDiagDataLogTime.wSecond+1;
			IF(stDiagDataLogTime.wSecond>=60)THEN
				stDiagDataLogTime.wSecond:=stDiagDataLogTime.wSecond-60;
				stDiagDataLogTime.wMinute:=stDiagDataLogTime.wMinute+1;
				IF(stDiagDataLogTime.wMinute>=60)THEN
					stDiagDataLogTime.wMinute:=stDiagDataLogTime.wMinute-60;
					stDiagDataLogTime.wHour:=stDiagDataLogTime.wHour+1;
				END_IF
			END_IF
		END_IF
		msecond:=msecond+LREAL_TO_WORD(MIN(MAX(1000.0*fCycleTime,1.0),30000.0));
		fbGetTime(START:=(msecond>1100));
		IF fbGetTime.START THEN
			IF(NOT fbGetTime.BUSY)THEN
				IF(fbGetTime.ERR)THEN
					msecond:=0;
				ELSE
					stDiagDataLogTime:=fbGetTime.TIMESTR;
					msecond:=fbGetTime.TIMESTR.wMilliseconds;
				END_IF
			END_IF
		END_IF

		CASE nWrState OF

			0:	IF bInputDoWrite THEN
					bBusyWriting:= TRUE;
					IF bDiagDataLogRunOn_WinCE THEN
						sWrite:=CONCAT(cnst_DiagDataLogFilePath_CE,cnst_SubDir_DiagDataLog);
					ELSE
						sWrite:=CONCAT(cnst_DiagDataLogFilePath_XP,cnst_SubDir_DiagDataLog);
					END_IF
					sWrite:=CONCAT(sWrite,cnst_FileName);
					stWrTime:=stDiagDataLogTime;
					stemp:=WORD_TO_STRING(stWrTime.wYear);
					stemp:=CONCAT(stemp,'_');
					IF(stWrTime.wMonth<10)THEN
						stemp:=CONCAT(stemp,'0');
					END_IF
					stemp:=CONCAT(stemp,WORD_TO_STRING(stWrTime.wMonth));
					stemp:=CONCAT(stemp,'_');
					IF(stWrTime.wDay<10)THEN
						stemp:=CONCAT(stemp,'0');
					END_IF
					stemp:=CONCAT(stemp,WORD_TO_STRING(stWrTime.wDay));
					stemp:=CONCAT(stemp,'_');
					IF(stWrTime.wHour<10)THEN
						stemp:=CONCAT(stemp,'0');
					END_IF
					stemp:=CONCAT(stemp,WORD_TO_STRING(stWrTime.wHour));
					stemp:=CONCAT(stemp,'.LOG');
					fbOpen.sPathName:=CONCAT(sWrite,stemp);
					fbOpen.bExecute:=FALSE;
					nWrState:=1;
				END_IF
	
			1:	fbOpen(sNetId:='', nMode:=FOPEN_MODEAPPEND OR FOPEN_MODETEXT, ePath:=PATH_GENERIC, tTimeout:=T#5S);
				IF NOT fbOpen.bExecute THEN
					fbOpen.bExecute:=TRUE;
				ELSIF NOT fbOpen.bBusy THEN
					IF fbOpen.bError THEN
						bInputDoWrite:=FALSE;
						nWrState:=0;
					ELSE
						fbWrite(sNetId:='', hFile:=fbOpen.hFile, pWriteBuff:=0, cbWriteLen:=0, bExecute:=FALSE, tTimeout:=T#5s);
						fbClose(sNetId:='', hFile:=fbOpen.hFile, bExecute:=FALSE, tTimeout:=T#5s);
						nWrState:=2;
					END_IF
					fbOpen(bExecute:=FALSE);
				END_IF

			2:	(**)
					stemp:=WORD_TO_STRING(stWrTime.wYear);
					stemp:=CONCAT(stemp,'.');
					IF(stWrTime.wMonth<10)THEN
						stemp:=CONCAT(stemp,'0');
					END_IF
					stemp:=CONCAT(stemp,WORD_TO_STRING(stWrTime.wMonth));
					stemp:=CONCAT(stemp,'.');
					IF(stWrTime.wDay<10)THEN
						stemp:=CONCAT(stemp,'0');
					END_IF
					stemp:=CONCAT(stemp,WORD_TO_STRING(stWrTime.wDay));
					stemp:=CONCAT(stemp,'|');
					IF(stWrTime.wHour<10)THEN
						stemp:=CONCAT(stemp,'0');
					END_IF
					stemp:=CONCAT(stemp,WORD_TO_STRING(stWrTime.wHour));
					stemp:=CONCAT(stemp,':');
					IF(stWrTime.wMinute<10)THEN
						stemp:=CONCAT(stemp,'0');
					END_IF
					stemp:=CONCAT(stemp,WORD_TO_STRING(stWrTime.wMinute));
					stemp:=CONCAT(stemp,':');
					IF(stWrTime.wSecond<10)THEN
						stemp:=CONCAT(stemp,'0');
					END_IF
					stemp:=CONCAT(stemp,WORD_TO_STRING(stWrTime.wSecond));
					stemp:=CONCAT(stemp,':');
					IF(stWrTime.wMilliseconds<10)THEN
						stemp:=CONCAT(stemp,'00');
					END_IF
					IF(stWrTime.wMilliseconds<100)
					AND stWrTime.wMilliseconds>=10 THEN
						stemp:=CONCAT(stemp,'0');
					END_IF
					stemp:=CONCAT(stemp,WORD_TO_STRING(stWrTime.wMilliseconds));
					stemp:=CONCAT(stemp,'|');

				sWriteData:=sWrite:=CONCAT(stemp , sActUseingString);
				sWrite:=CONCAT(sWrite,'$n');
				fbWrite(pWriteBuff:=ADR(sWrite), cbWriteLen:=LEN(sWrite), bExecute:=TRUE);
				nWrState:=3;

			3:	fbWrite(pWriteBuff:=ADR(sWrite), cbWriteLen:=LEN(sWrite), bExecute:=TRUE);
				IF NOT fbWrite.bBusy THEN
					IF fbWrite.bError THEN
						nWrState:=-4;
					ELSE
						nWrState:=10;
					END_IF
					fbWrite(bExecute:=FALSE);
				END_IF

			-4,
			10:fbClose(bExecute:=TRUE);
				IF NOT fbClose.bBusy THEN
					IF fbClose.bError THEN
						bBusyWriting:=FALSE;
						bInputDoWrite:=FALSE;
						nWrState:=0;
					ELSE
						bBusyWriting:=FALSE;
						bInputDoWrite:=FALSE;
						nWrState:=0;
					END_IF
					fbClose(bExecute:=FALSE);
				END_IF
		END_CASE
	END_IF



END_CASE
END_ACTION

ACTION act_CheckCom:


	IF sInputString<>''(*ÓÐÐÂµÄ¼ÇÂ¼ÐèÒªÐ´*)
	AND nState=11 THEN
		FOR i:=1 TO 10 DO
			IF aStringBuffer[i]='' THEN
				aStringBuffer[i]:=sInputString;(*·Åµ½»º´æ*)
				EXIT;
			END_IF
		END_FOR
		sInputString:='';
	END_IF

	IF aStringBuffer[1]<>''(*»º´æÓÐÐèÒªÐ´µÄ¼ÇÂ¼*)
	AND NOT bInputDoWrite THEN
		sActUseingString:=aStringBuffer[1];
		FOR i:=1 TO 9 DO
			aStringBuffer[i]:= aStringBuffer[i+1];
		END_FOR
		aStringBuffer[10]:='';
		bInputDoWrite:=TRUE;
	END_IF
END_ACTION

ACTION act_Copy2USB:

(*¸´ÖÆµ½ÆäËüÎÄ¼þ¼Ð*)
CASE CopyStep OF
	0:
		IF bCopyToUSB THEN
			CopyStep:=100;
		END_IF

	100:
		IF bDiagDataLogRunOn_WinCE THEN
			fbDirectoryCopy.srcPathName:=cnst_DiagDataLogFilePath_CE;
			fbDirectoryCopy.destPathName:=cnst_USB_FilePath_CE;
		ELSE
			fbDirectoryCopy.srcPathName:=cnst_DiagDataLogFilePath_XP;
			fbDirectoryCopy.destPathName:=cnst_USB_FilePath_XP;
		END_IF
		fbDirectoryCopy.DirectoryName:= LEFT(cnst_SubDir_DiagDataLog,LEN(cnst_SubDir_DiagDataLog)-1);
		fbDirectoryCopy.FileType:= 		'log';
		CopyStep:=200;

	200:
		fbDirectoryCopy(bExecute:=TRUE);
		IF fbDirectoryCopy.bBusy THEN
			CopyStep:=300;
		END_IF

	300:
		fbDirectoryCopy();
		IF NOT fbDirectoryCopy.bBusy THEN
			fbDirectoryCopy(bExecute:=FALSE);
			CopyStep:=400;
		END_IF

	400:
		IF NOT bCopyToUSB THEN
			CopyStep:=0;
		END_IF

END_CASE
END_ACTION

END_FUNCTION_BLOCK

// ---- DUTs/文件配方/Swen_Products/FB_DirectoryCopy.TcPOU
FUNCTION_BLOCK FB_DirectoryCopy
(*SwenChen 2011.4.13 编辑*)
VAR_INPUT
	srcNetId				: T_AmsNetId;	(* TwinCAT network address of the source file *)
	srcPathName			: T_MaxString;	(* source file path *)(*源的地址*)
	destNetId			: T_AmsNetId;	(* TwinCAT network address of the destination file *)
	destPathName		: T_MaxString;  	(* destination file path  *)(*目标的上层地址*)
	DirectoryName		: T_MaxString;  	(* destination file  name *)(*目标文件夹名字*)
	FileType				: STRING:='*';  		(* destination file  name *)(*文件类型*)
	bExecute			: BOOL;			(* rising edge start fb execution *)
	bFindFileList			: BOOL;			(* rising edge start fb execution *)
	tAdsTimeOut			: TIME;			(* ads timeout *)
	bContinueWhenErr	:BOOL;
	bCancelWhenErr		:BOOL;
END_VAR
VAR_OUTPUT
	bBusy				:BOOL;
	bError				:BOOL;
	nErrId				:UDINT;
	(*==============
	ErrId:=1;		(*ErrId: no find source dir*)
	ErrId:=2;		(*ErrId: no find target dir*)
	ErrId:=3:		target have same file;
	ErrId:=4:		(*Input parameter error*)
	================*)
END_VAR
VAR
	Step				:DWORD;
	RisingEdge			:R_TRIG;
	fbFindFileList:			FB_EnumFindFileList;
	fbEnumFindFileEntry:	FB_EnumFindFileEntry;
	srcFilesLists:			 ARRAY[1..12]  OF ST_FindFileEntry;
	destFilesLists:		 ARRAY[1..12]  OF ST_FindFileEntry;
	fbFileCopy:			FB_FileCopy;
	fbCreateDir:			FB_CreateDir;
	i: 					INT;
	n:					INT;
	bFindFileListState		: BOOL;
	TimeCount:			 INT;
END_VAR

RisingEdge(CLK:=bExecute OR bFindFileList);

IF bBusy THEN
	TimeCount:=TimeCount+1;
END_IF

CASE Step OF
	0:	(* do nothing *)
		IF RisingEdge.Q  AND NOT bBusy THEN
			IF bFindFileList THEN
				bFindFileListState:=TRUE;
				bBusy := TRUE;
				Step := 40;
			ELSE
				bFindFileListState:=FALSE;
				IF DirectoryName=''
				OR FileType=''
				OR srcPathName=''
				OR destPathName='' THEN		(*Input parameter error*)
					bError:=TRUE;
					nErrId:=4;
				ELSE
					bBusy := TRUE;
					bError:= FALSE;
					TimeCount:=0;
					nErrId:=0;
					Step := 10;
				END_IF
			END_IF
		END_IF

	10:	(* find source dir*)
		fbEnumFindFileEntry
			(
			sNetId:='' , 
			sPathName:=CONCAT(srcPathName,DirectoryName),
			eCmd:=eEnumCmd_First ,
			bExecute:=TRUE ,
			tTimeout:=T#10s ,
			);
		IF NOT  fbEnumFindFileEntry.bBusy THEN
			IF NOT  fbEnumFindFileEntry.bEOE THEN		(*target dir is exist*)
				Step := 20;
			ELSE										(*target dir no exist*)
				bError:=TRUE;
				nErrId:=1;		(*ErrId: no find source dir*)
				Step:=70;
			END_IF
			fbEnumFindFileEntry(bExecute:=FALSE);
		END_IF

	11:	(*Wait*)
		IF bContinueWhenErr OR bCancelWhenErr THEN
			bError:=FALSE;
			nErrId:=0;
			Step:=0;
		END_IF

	20:	(*find Target Dir*)
		fbEnumFindFileEntry
			(
			sNetId:='' , 
			sPathName:=CONCAT(destPathName,DirectoryName),
			eCmd:=eEnumCmd_First ,
			bExecute:=TRUE ,
			tTimeout:=T#10s ,
			);
		IF NOT  fbEnumFindFileEntry.bBusy THEN
			IF NOT  fbEnumFindFileEntry.bEOE THEN	(*target dir is exist*)
				Step := 40;
			ELSE									(*target dir no exist*)
				Step:=30;
			END_IF
			fbEnumFindFileEntry(bExecute:=FALSE);
		END_IF

	30:	(*createt dir  *)
		fbCreateDir
			(
			sNetId:='',
			sPathName:= CONCAT(destPathName,DirectoryName),
			ePath:= PATH_GENERIC,
			bExecute:=TRUE,
			tTimeout:=t#10s
			);
		IF NOT fbCreateDir.bBusy THEN
			fbCreateDir(bExecute:=FALSE);
			Step:=40;
		END_IF

	40:	(*Find source FileList*)
		fbFindFileList
			(
			sNetID:='',
			sPathName:=CONCAT(CONCAT(CONCAT(srcPathName,DirectoryName),'\*.'),FileType),
			eCmd:= eEnumCmd_First,
			pFindList:= ADR(srcFilesLists),
			cbFindList:=SIZEOF(srcFilesLists),
			bExecute:= TRUE ,
			tTimeout:=t#10s
			);
		IF NOT fbFindFileList.bBusy THEN
			fbFindFileList(bExecute:=FALSE);
			IF bFindFileList OR bFindFileListState THEN
				Step:=70;
			ELSE
				Step:=41;
			END_IF
		END_IF

	41:	(*Find target FileList*)
		fbFindFileList
			(
			sNetID:='',
			sPathName:=CONCAT(CONCAT(CONCAT(destPathName,DirectoryName),'\*.'),FileType),
			eCmd:= eEnumCmd_First,
			pFindList:= ADR(destFilesLists),
			cbFindList:=SIZEOF(destFilesLists),
			bExecute:= TRUE ,
			tTimeout:=t#10s
			);
		IF NOT fbFindFileList.bBusy THEN
			fbFindFileList(bExecute:=FALSE);
			Step:=50;
			i:=1;
		END_IF


	50:	(*check no same mane file*)
		IF srcFilesLists[i].sFileName='' THEN
			IF i>=15 THEN
				i:=1;
				Step:=70;
			ELSE
				i:=i+1;
			END_IF
		ELSE
			FOR n:=1 TO 15 DO
				IF destFilesLists[n].sFileName =  srcFilesLists[i].sFileName THEN
					bError:=TRUE;
					nErrId:=3;
				END_IF
			END_FOR
			IF  bError THEN			(*if exiest same file *)
				IF bContinueWhenErr THEN
					Step:=60;
					bError:=FALSE;
					nErrId:=0;
				ELSIF bCancelWhenErr THEN
					i:=i+1;
					bError:=FALSE;
					nErrId:=0;
				END_IF
			ELSE					(*no same file *)
				fbFileCopy
					(
					srcNetId:='' ,
					srcFileName:=CONCAT(CONCAT(CONCAT(srcPathName,DirectoryName),'\'),srcFilesLists[i].sFileName) ,
					cbReadLen:=srcFilesLists[i].fileSize.dwLowPart,
					destNetId:='' ,
					destFileName:=CONCAT(CONCAT(CONCAT(destPathName,DirectoryName),'\'),srcFilesLists[i].sFileName) ,
					bExecute:=TRUE ,
					tAdsTimeOut:=T#10s ,
					);
				Step:=60;
			END_IF
		END_IF

	60:	(*copy*)
		fbFileCopy();
		IF NOT fbFileCopy.bBusy THEN
			fbFileCopy(bExecute:=FALSE);
			IF i>=15 THEN
				i:=1;
				Step:=70;
			ELSE
				i:=i+1;
				Step:=50;
			END_IF
		END_IF

	70:	(*finish*)
		bFindFileListState:=FALSE;
		bBusy := FALSE;
		Step:=0;

END_CASE

END_FUNCTION_BLOCK

// ---- DUTs/文件配方/Swen_Products/FB_FileCopy.TcPOU
FUNCTION_BLOCK FB_FileCopy
(*SwenChen 2011.4.13 修改于帮助文件*)
VAR_INPUT
	srcNetId				: T_AmsNetId;	(* TwinCAT network address of the source file *)
	srcFileName			: T_MaxString;	(* source file path and name *)
	destNetId			: T_AmsNetId;	(* TwinCAT network address of the destination file *)
	destFileName		: T_MaxString;  (* destination file path and name *)
	bExecute			: BOOL;			(* rising edge start fb execution *)
	tAdsTimeOut			: TIME;			(* ads timeout *)
	cbReadLen			: UDINT;
END_VAR
VAR_OUTPUT
	bBusy				:BOOL;
	bError				:BOOL;
	nErrId				:UDINT;
END_VAR
VAR
	fbFileOpen			:FB_FileOpen;
	fbFileClose			:FB_FileClose;
	fbFileRead			:FB_FileRead;
	fbFileWrite			:FB_FileWrite;

	hSrcFile				:UINT	:= 0;(* file handle of the source file *)
	hDestFile			:UINT	:= 0;(* file handle of the destination file *)

	Step				:DWORD;
	RisingEdge			:R_TRIG;

	buffRead				:ARRAY[1..30000] OF BYTE;(* buffer *)
	cbReadLength		:UDINT:=0;
	TimeCount			:INT;
END_VAR

RisingEdge(CLK:=bExecute);
IF RisingEdge.Q THEN
	IF NOT bBusy THEN
		bBusy := TRUE;
		bError:= FALSE;
		nErrId:=0;
		Step := 1;
		cbReadLength:=0;
		hSrcFile:=0;
		hDestFile:=0;
		TimeCount:=0;
	END_IF
END_IF

IF bBusy THEN
	TimeCount:=TimeCount+1;
END_IF


CASE Step OF
	0:	(* do nothing *)
		;

	1:	(* open source file *)
		fbFileOpen(  bExecute := FALSE  );
		fbFileOpen( 	sNetId := srcNetId,
						sPathName := srcFileName,
						nMode := FOPEN_MODEREAD OR FOPEN_MODEBINARY(*FOPEN_MODETEXT*),
						ePath := PATH_GENERIC,
						tTimeout := tAdsTimeout,
						bExecute := TRUE );
		Step := Step + 1;

	2:
		fbFileOpen( bExecute := FALSE );
		IF ( NOT fbFileOpen.bBusy ) THEN
			IF ( fbFileOpen.bError ) THEN
				nErrId := fbFileOpen.nErrId;
				bError := TRUE;
				Step := 50;
			ELSE
				hSrcFile := fbFileOpen.hFile;
				Step := Step + 1;
			END_IF
		END_IF

	3:	(* open destination file *)
		fbFileOpen(  bExecute := FALSE  );
		fbFileOpen( 	sNetId := destNetId,
						sPathName := destFileName,
						nMode := FOPEN_MODEWRITE OR FOPEN_MODEBINARY(*FOPEN_MODETEXT*),
						ePath := PATH_GENERIC,
						tTimeout := tAdsTimeout,
						bExecute := TRUE );
		Step := Step+1;

	4:
		fbFileOpen(  bExecute := FALSE  );
		IF ( NOT fbFileOpen.bBusy ) THEN
			IF ( fbFileOpen.bError ) THEN
				nErrId := fbFileOpen.nErrId;
				bError := TRUE;
				Step := 50;
			ELSE
				hDestFile := fbFileOpen.hFile;
				Step := Step + 1;
			END_IF
		END_IF

	5:	(*read data from source file*)
		cbReadLength := 0;
		fbFileRead( bExecute:= FALSE );
		fbFileRead( 	sNetId:=SrcNetId,
						hFile:=hSrcFile,
						pReadBuff:= ADR(buffRead),
						cbReadLen:= (*SIZEOF(buffRead)*)cbReadLen,
						bExecute:=TRUE,
						tTimeout:=tAdsTimeOut );
		Step := Step + 1;

	6:
		fbFileRead( bExecute:= FALSE );
		IF ( NOT fbFileRead.bBusy ) THEN
			IF ( fbFileRead.bError ) THEN
				nErrId := fbFileRead.nErrId;
				bError := TRUE;
				Step := 50;
			ELSE
				cbReadLength := fbFileRead.cbRead;
				Step := Step + 1;
			END_IF
		END_IF

	7:	(*write data to destination file*)
		fbFileWrite( bExecute := FALSE );
		fbFileWrite(	sNetId:=DestNetId,
						hFile:=hDestFile,
						pWriteBuff:= ADR(buffRead),
						cbWriteLen:= cbReadLength,
						bExecute:=TRUE,
						tTimeout:=tAdsTimeOut );
		Step := Step + 1;

	8:
		fbFileWrite( bExecute := FALSE );
		IF ( NOT fbFileWrite.bBusy ) THEN
			IF ( fbFileWrite.bError ) THEN
				nErrId := fbFileWrite.nErrId;
				bError := TRUE;
				Step := 50;
			ELSE
				IF fbFileRead.bEOF THEN (*Check if the EOF flag ist set *)
					Step := 50;		(*cleanup: close the destination and source files *)
				ELSE
					Step := 5; (* repeat reading *)
				END_IF
			END_IF
		END_IF

	30:	(* close the destination file *)
		fbFileClose( bExecute := FALSE );
		fbFileClose( 	sNetId:=destNetId,
						hFile:=hDestFile,
						bExecute:=TRUE,
						tTimeout:=tAdsTimeOut );
		Step := Step + 1;

	31:
		fbFileClose( bExecute := FALSE );
		IF ( NOT fbFileClose.bBusy ) THEN
			IF ( fbFileClose.bError ) THEN
				nErrId := fbFileClose.nErrId;
				bError := TRUE;
			END_IF
			Step := 50;
			hDestFile := 0;
		END_IF

	40: (* close source file *)
		fbFileClose( bExecute := FALSE );
		fbFileClose( 	sNetId:=srcNetId,
						hFile:=hSrcFile,
						bExecute:=TRUE,
						tTimeout:=tAdsTimeOut );
		Step := Step + 1;

	41:
		fbFileClose( bExecute := FALSE );
		IF ( NOT fbFileClose.bBusy ) THEN
			IF ( fbFileClose.bError ) THEN
				nErrId := fbFileClose.nErrId;
				bError := TRUE;
			END_IF
			Step := 50;
			hSrcFile := 0;
		END_IF

	50: (*error or ready => cleanup*)
		IF ( hDestFile <> 0 ) THEN
			Step := 30; (* close the destination file*)
		ELSIF (hSrcFile <> 0 ) THEN
			Step := 40; (* close the source file *)
		ELSE
			Step := 0;	(* ready *)
			bBusy := FALSE;
		END_IF

END_CASE

END_FUNCTION_BLOCK

// ---- POUs/EventGridTest/EventGrid.TcPOU
PROGRAM EventGrid
VAR
	fbEventlogger : FB_TcEventLogger;
	fbAlarm: FB_TcAlarm;
	fbMessage: FB_TcMessage;
	bAlarm: BOOL;
	bMessage : BOOL;
	bIsInitalized: BOOL;
	bClearAlarm: BOOL;
	bConfirmAlarm: BOOL;
END_VAR

IF NOT bIsInitalized THEN
	bIsInitalized := TRUE;
	fbMessage.CreateEx(TC_Events.Sinterstar_Mini_EventClass.Sinterstar_Mini_EventClassEvent2, 0);
	fbAlarm.CreateEx(TC_Events.Sinterstar_Mini_EventClass.Sinterstar_Mini_EventClassEvent2, TRUE, 0);
END_IF

IF bMessage THEN
	bMessage := FALSE;
	fbMessage.Send(0);
END_IF

IF bAlarm THEN
	bAlarm := FALSE;
	fbAlarm.Raise(0);
END_IF

IF bClearAlarm THEN
	bClearAlarm := FALSE;
	fbAlarm.Clear(0, FALSE);
END_IF

END_PROGRAM

// ---- POUs/Line_chart.TcPOU
PROGRAM Line_chart
VAR
	aPoints : ARRAY [1..2,1..10000] OF ST_Point;
	bInit : BOOL := TRUE;
	nCounter: INT:=10000;
	nValue1 : INT := 1;
	nValue2 : INT := -1;
	btag1: BOOL;
	i: INT;
	nposrang: INT:=10000;
	tTimer: ToN;
	nsamptime	:TIME:=T#50MS;
	bstart: BOOL;
	tTimer1: TON;
	Et1: TIME;
	Tnow_time: REAL;
	sin_n_int: LREAL;
	sin_n:LREAL;
	bclear: BOOL;
	AMP:INT:=10;
END_VAR

IF bInit THEN
	FOR nCounter := 1 TO 10000 DO
		aPoints[1, nCounter].x := nCounter;// nCounter
		//aPoints[2, nCounter].x := nCounter;
		aPoints[2, nCounter].y := 1000;
	END_FOR
	
		bInit := FALSE;
END_IF
IF NOT btag1 THEN
	
	FOR i:=nposrang TO 1 BY -1 DO
	aPoints[1, nposrang].y :=0;
	aPoints[1, nposrang].x :=0;
	END_FOR
	btag1:=TRUE;
ELSE
	tTimer(IN:=NOT tTimer.q , PT:=nsamptime , Q=> , ET=> );
IF bstart THEN
	tTimer1(IN:=NOT tTimer1.q , PT:=T#10D , Q=> , ET=>Et1 );
	Tnow_time:=TIME_TO_REAL(Et1)/1000;
END_IF
bstart:=main.bStartTemControl;
IF tTimer.Q AND bstart THEN
	sin_n_int:=sin_n_int+0.005;
	sin_n:=SIN(pi*sin_n_int)*AMP;
	//目标数据采集
FOR nCounter:=nposrang TO 2 BY -1 DO	
	aPoints[1, nCounter].y := aPoints[1, nCounter - 1].y;
	aPoints[1, nCounter].x := aPoints[1, nCounter - 1].x;
END_FOR
	aPoints[1, 1].y := Controller_v2.ftemp_convert;//Controller_v2.ftemp
	aPoints[1, 1].x := Tnow_time;
END_IF
END_IF
IF bclear THEN 						//清空数据
	FOR nCounter := 1 TO 1000  DO
	aPoints[1, nCounter].x :=0;
	aPoints[1, nCounter].y :=0;
	//sin_n_int:=0;
	END_FOR
END_IF

END_PROGRAM

// ---- POUs/Controller_v2.TcPOU
PROGRAM Controller_v2

VAR
		iTempre_Compare			AT %I*:INT;   
		fTempre_Actual			:LREAL; 
		fTempre_Actual_convert	:LREAL; 
		itest					:LREAL; 
		eCTRL_Mode 				: E_CTRL_MODE := eCTRL_MODE_Tune; 	(*控制模式*)
		bSelSetpoint			: BOOL	:= FALSE;
		
			iTempre AT %I*:INT;                                  (* 传输回未被转换的温度值 *)
			ftemp :LREAL;                                         (* 被转换的实际温度值 *)
		ftemp_convert	:LREAL; 
		fW						: LREAL;						(* 设定值 *)
		
		fY						: LREAL;						(* 模拟量输出中间变量 *)
		fX						: LREAL;						(* 设备真实的温度值 *)
		bYPWMPos				AT %Q*: BOOL;                   (* PWM输出，加热 *)
		bYPWMNeg				AT %Q*: BOOL;                   (* PWM输出，冷却 *)
		
		bNoise					: BOOL;                         (* 系统中是否存在错误 *)
		bError 					: BOOL;                         (* 存在错误的话，会生成一个错误代码 *)
		eErrorId 				: E_CTRL_ErrorCodes;
		
		stControllerParameter	: ST_CTRL_TempCtrlParameter := (		
		
		(*内部结构体参数 *)
		iMode					:= 1,											(*运作模式 ： 1=加热, 2=冷却, 3=加热以及冷却 *)
		iReactionOnFailure		:= eCTRL_ReactionOnFailure_StopController,		(*当系统产生错误时，系统反应： 0=关闭系统, 1=手动操作 *)
	
		bSelCtrlParameterSet	:= FALSE,										(* FALSE = 内部pid设定, TRUE = 外部pid设定 *)
	
		dwAlarmSupp				:= 16#0000EFFF,									(* 报警限制值 *)
		tCtrlCycleTime			:= T#500MS,										(* 控制器周期时间 *)
		tTaskCycleTime			:= T#10MS,										(* PLC任务周期时间 *)
		
		(*整定参数*)
		iTuningMode				:= 1,											(* 只加热、只冷却、先加热后冷却、先冷却后加热 *)
	
		tTuneStabilisation		:= T#5S,										(* 等待系统稳定下的时间 *)
	
		fEndTunePercentHeating	:= 80.0,										(* 大于80%，切换成闭环控制 *)
		fYTuneHeating			:= 100.0,										(* 加热协调操作时的阶跃变换 *)
		fYStableHeating			:= 0.0,											(* 加热调整操作 *)
	
		fEndTunePercentCooling	:= 20.0,										(* 小于20%，切换成闭环控制 *)
		fYTuneCooling			:= 0.0,									        (*冷却协调操作时的阶跃变换 *)
		fYStableCooling			:= 0.0,											(* 冷却调整操作 *)
		fScalingFactor			:= 1.0,											(*加热和冷却的KP比例系数 *)
		
		(*设定点参数*)
		fWMin					:= 0.0,											(*设定点的最小值 *)
		fWMax					:= 300.0,										(*设定点的最大值 *)
	
		(*软启动*)
		bEnableSoftStart		:= TRUE,										(* 启动方式：FALSE = 硬启动, TRUE = 软启动 *)
		bEnableRamping			:= FALSE,										(* 波形：FALSE = 无斜波, TRUE = 有斜波 *)
	
		fWStartUp				:= 55.0,										(* 软启动的预设定值 *)
		tStartUp				:= T#30S,										(* 软启动的等待时间*)
		bStartUpRamping			:= FALSE,										(* 启动过程时是否加入斜波 *)
		fWStartUpVeloPos		:= 0.3,											(* 启动过程时增加给定的最大梯度值*)
		fWStartUpVeloNeg		:= 0.3,											(* 启动过程时减小给定的最大梯度值 *)
	
		fWVeloPos				:= 0.5,											(* 增加给定的最大梯度值 *)
		fWVeloNeg				:= 0.5,											(* 减小给定的最大梯度值 *)	
	
		(* 实际值参数*)
		bFilter 				:= FALSE,                                       (* 是否启动实际值过滤器*)
		tFilter					:= T#0S,                                        (* 实际值过滤器的时间常数*)
		
		(* 死区参数 *)
		bDeadband				:= FALSE,                                       (* 是否加入死区 *)
		fEDeadband				:= 0.0,											(* 死区参数 *)
		
		(* 控制值参数*)
		fYMin					:= 0.0,											(* 控制器下限值 *)
		fYMax					:= 100.0,										(* 控制器上限值 *)
		fYManual				:= 0.0,									 		(* 手动操作值*)
		fYOnFailure				:= 0.0,											(* 故障时的手动控制值 *)
		tPWMCycleTime			:= T#1S,										(* PWM周期 *)
		tPWMMinOffTime			:= T#0S,										(* PWM最小的关闭时间*)
		tPWMMinOnTime			:= T#0S,										(* PWM最小的开启时间 *)
		tPWMWaitingTime			:= T#0S,										(* PWM从加热到冷却的切换时间*)
		tPWMCycleTimeCool       := T#1S,                                        (* PWM冷却周期 *)
	
		fYThresholdOff			:= 0.0,											(* 三步关闭极限，此例程不需要使用 *)
		fYThresholdOn			:= 0.0,											(* 三步开启极限，此例程不需要使用 *)
	
		nCyclesForSwitchOver	:= 100,                                         (* 参数级转换数 *) 
	
		(* 控制器设定 *)
		bEnablePreController 	:= FALSE,										(* 允许预控制器 *)
		bEnableZones 			:= FALSE,										(* 允许开环调节时的设定调节带 *)
		bEnableCVFilter 		:= FALSE,										(* 允许CV滤波 *)
		iFilterType 			:= 1,			 			                    (* CV滤波器类型，系统默认设定 *)
		iControllerType 		:= eCTRL_ControllerType_PID,					(* 控制器的PID类型，系统默认设定 *)
		
		
		(* 最小最大温度 *) 
		TempLow					:= -5.0,                                        (* 第一道报警值下限 *) 
		TempLowLow				:= -10.0,                                       (* 第二道报警值下限 *)
		TempHigh				:= 80.0,                                        (* 第一道报警值上限 *)
		TempHighHigh			:= 100.0,                                       (* 第二道报警值上限 *)
		TempAbsoluteHigh		:= 300.0,                                       (* 设定报警值上限 *)
		TempAbsoluteLow			:= 0.0,	                                        (* 设定报警值下限 *)
		
		(* 内部整定高级参数 *)
		fTuneKp					:= 1.0,                                         (* 比例 *)
		fTuneTn					:= 2.5,                                         (* 积分时间常数 *)
		fTuneTv					:= 0.42,                                        (* 微分时间常数 *)
		fTuneTd					:= 0.25                                         (* 阻尼时间常数 *)
		);
	
	fbTempController			: FB_CTRL_TempController;                       (* 功能块声明 *)
	

	fbCtrlParameter				: FB_CTRL_CtrlParameter;                        (* 功能块声明 *)
	stController				: ST_CTRL_ParaController;                       (* 结构体变量声明 *)
	fbgetinfo					:FB_GetAdaptersInfo;

	Address						:ARRAY[0..MAX_LOCAL_ADAPTERS]OF ST_IpAdapterInfo;
	NetID: T_AmsNetId:='';
	bExecute: BOOL;
	bHeater_2 AT%Q*: BOOL;
END_VAR
VAR PERSISTENT
fW1						: LREAL ;				(* 主设定值(保温值)*)
fW2						: LREAL ;				(* 辅助设定值(加热值)*)		

END_VAR

fbgetinfo(
	sNetID:= '5.127.65.238.1.1', 
	bExecute:= bExecute, 
	tTimeout:= , 
	bBusy=> , 
	bError=> , 
	nErrID=> , 
	arrAdapters=>Address , 
	nCount=> , 
	nGet=> );
(* 接收的温度数据转换 *)
fTempre_Actual:=INT_TO_LREAL(iTempre_Compare);
fTempre_Actual_convert:=fTempre_Actual/10;
ftemp:=INT_TO_LREAL (iTempre);
ftemp_convert:=ftemp/10;
(* 选择设定点 *)
IF bSelSetpoint THEN
	fW := fW2;
ELSE
	fW := fW1;
END_IF


(* 实际温度值中间变量转换*)				
fbTempController.fX:=ftemp;		

(* 设置功能块参数，只需修改 fX:=ftemp *)
fbTempController(
					eCtrlMode				:= eCTRL_Mode, 
					bSelSetpoint			:= bSelSetpoint, 
					fW1						:= fW1, 	//保温值
					fW2						:= fW2, 	//一阶加温值
					fX						:= ftemp_convert, //反馈温度
					fYManual				:= , 
					bOpenThermocouple		:= FALSE, 
					bReverseThermocouple	:= FALSE, 
					bBackVoltage			:= FALSE, 
					bLeakage				:= FALSE, 
					bShortCircuit			:= FALSE, 
					bOpenCircuit			:= FALSE, 
					sParaControllerExternal	:= stController, 
					sControllerParameter	:= stControllerParameter, 
					);
					 
(* 模拟量输出，此例程无需使用 *)			
//fY := fbTempController.fYAnalog;
//IF  NOT main.bStartTemControl THEN
//	bYPWMPos :=FALSE;
//END_IF
(* PWM加热输出 *)
bYPWMPos := fbTempController.bYPWMPos;
bHeater_2:=	fbTempController.bYPWMPos;
(* PWM冷却输出，此例程无需使用 *)
//bYPWMNeg := fbTempController.bYPWMNeg;

bError := fbTempController.bError;
eErrorId := fbTempController.eErrorId;

(* 选择控制器模式。第一次使用时，eCTRL_Mode必须先进入自整定模式：eCTRL_STATE_TUNED 进行参数整定的操作*)
(* 参数整定之后，再进入主动模式使系统控制温度 *)
IF fbTempController.eCtrlState = eCTRL_STATE_TUNED THEN
	eCTRL_Mode := eCTRL_MODE_ACTIVE;	
END_IF

END_PROGRAM

// ---- POUs/文件记录/data_save.TcPOU
PROGRAM data_save
VAR
	T_heat			:INT;
	
	fbSysTime		:GETSYSTEMTIME;
	tFileTime		:T_FILETIME;  	
	tNow			:TIMESTRUCT; 
	fbFormatString 	:FB_FormatString;
	fbFormatString1	:FB_FormatString;
	tNowTime		:T_MaxString ;
	sPathFormat		:T_MaxString := '%s\%d__%d_%d_%d_%d_%d.csv';	
	tTimeFormat		:T_MaxString := '%d__%d_%d_%d_%d_%d';		
	wHour: WORD;
	sPath: STRING(255);
	bWrite			:BOOL;//写入触发
	sNetId			: T_AmsNetId := '';	
	sFileName		: T_MaxString ;
	sCSVLine		: T_MaxString := '';
	sCSVField		: T_MaxString := '';
	bBusy			: BOOL;
	bError			: BOOL;
	nErrId			: UDINT;
	nRow	 		: UDINT 	:= 0;
	nColumn			: UDINT 	:= 0;
	hFile			: UINT		:= 0;
	step			: DWORD 	:= 0;
	fbFileOpen		: FB_FileOpen;
	fbFileClose		: FB_FileClose;
	fbFilePuts		: FB_FilePuts;
	fbWriter		: FB_CSVMemBufferWriter;
	database		: ARRAY[0..MAX_CSV_ROWS, 0..MAX_CSV_COLUMNS ] OF STRING(MAX_CSV_FIELD_LENGTH);
	fbCycletime		:TON;
	rCurrentMaster		:LREAL;
	rTorque			:LREAL;
	rSpeed			:LREAL;
END_VAR
VAR CONSTANT
	tSamplefrequency:TIME:=T#1S;
	MAX_CSV_ROWS 			: UDINT :=600;//写入最大行数
	MAX_CSV_COLUMNS 		: UDINT :=3;	//写入最大列数0~3
	MAX_CSV_FIELD_LENGTH	: UDINT :=20000;
END_VAR

DEFAULT_CSV_FIELD_SEP := 16#2C;
fbSysTime(timeLoDW=>tFileTime.dwLowDateTime , timeHiDW=> tFileTime.dwHighDateTime);
tNow := FILETIME_TO_SYSTEMTIME(tFileTime);
wHour:=tNow.wHour+8;
sPath:='C:\Users\Administrator\Desktop\Temperature';
T_heat:=REAL_TO_INT(Line_chart.Tnow_time);

fbFormatString(
	sFormat:=sPathFormat, 
	arg1:=F_STRING(sPath) , 
	arg2:= F_WORD(tNow.wYear), 
	arg3:= F_WORD(tNow.wMonth), 
	arg4:= F_WORD(tNow.wDay), 
	arg5:= F_WORD(wHour), 
	arg6:= F_WORD(tNow.wMinute), 
	arg7:= F_WORD(tNow.wSecond),  
	sOut=> sFileName);
fbFormatString1(
	sFormat:=tTimeFormat, 
	//arg1:=F_STRING(sPath) , 
	arg1:= F_WORD(tNow.wYear), 
	arg2:= F_WORD(tNow.wMonth), 
	arg3:= F_WORD(tNow.wDay), 
	arg4:= F_WORD(wHour), 
	arg5:= F_WORD(tNow.wMinute), 
	arg6:= F_WORD(tNow.wSecond),  
	sOut=> tNowTime);	
IF tNow.wYear = 0 THEN
	RETURN;
END_IF
IF main.clk1.Q THEN
bWrite:=TRUE;
END_IF
CASE step OF
0:
IF bWrite THEN
	bWrite 	:= FALSE;
	bBusy 	:= TRUE;
	bError	:= FALSE;
	nErrId	:= 0;
	hFile	:= 0;
	nRow	:= 0;
	nColumn	:= 0;
	step 	:= 1;
END_IF
1:
	fbFileOpen(  bExecute := FALSE  );
	fbFileOpen( sNetId := sNetId, sPathName := sFileName, nMode := FOPEN_MODEWRITE OR FOPEN_MODETEXT,
				ePath := PATH_GENERIC, bExecute := TRUE );
	step := 2;
2:
	fbFileOpen( bExecute := FALSE, bError => bError, nErrID => nErrID, hFile => hFile );//err_ID 1804无法找到存储路径
IF NOT fbFileOpen.bBusy THEN
IF NOT fbFileOpen.bError THEN
	step := 3;
ELSE
	step := 100;
END_IF
END_IF
3:
IF NOT fbCycletime.Q AND main.bStartTemControl THEN
	fbCycletime(IN:=TRUE , PT:=tSamplefrequency , Q=> , ET=> );
ELSE 
IF nRow<>0 AND main.bStartTemControl THEN
	fbCycletime(IN:=FALSE , PT:=tSamplefrequency , Q=> , ET=> );
	sCSVLine := '';
	fbWriter.eCmd := eEnumCmd_First;
IF nRow <= MAX_CSV_ROWS AND main.bStartTemControl THEN
FOR nColumn:=0 TO MAX_CSV_COLUMNS BY 1 DO
	database[nRow,0]:=LREAL_TO_STRING(T_heat);//raw data
	database[nRow,1]:=LREAL_TO_STRING(Tem_Act_1);
	database[nRow,2]:=LREAL_TO_STRING(Tem_control_1);
	database[nRow,3]:=tNowTime;		//LREAL_TO_STRING(tNow.wSecond);
	sCSVField := STRING_TO_CSVFIELD( database[ nRow, nColumn ], FALSE );
	fbWriter( 	pBuffer := ADR( sCSVLine ), 
				cbBuffer := SIZEOF( sCSVLine ) - 1,
				putValue := sCSVField,
				pValue := 0, 
				cbValue := 0,
				bCRLF := ( nColumn = MAX_CSV_COLUMNS ) );
IF fbWriter.bOk THEN
	fbWriter.eCmd := eEnumCmd_Next;
ELSE
	step := 100;
RETURN;
END_IF
IF RIGHT( sCSVLine, 2 ) = '$R$L' THEN
	sCSVLine := REPLACE( sCSVLine, '$L', 2, LEN( sCSVLine ) - 1 );
END_IF	
END_FOR
	nRow := nRow + 1;
	step := 4;
ELSE
	step := 10;
END_IF
ELSE
	sCSVLine := '';
	fbWriter.eCmd := eEnumCmd_First;
	database[0,0]:='HeatingTime';
	database[0,1]:='Compare_Tem';
	database[0,2]:='Control_Tem';
	database[0,3]:='Time';
FOR nColumn:=0 TO MAX_CSV_COLUMNS BY 1 DO
	sCSVField := STRING_TO_CSVFIELD( database[ nRow, nColumn ], FALSE );
	fbWriter( 	pBuffer := ADR( sCSVLine ), 
				cbBuffer := SIZEOF( sCSVLine ) - 1, 
				putValue := sCSVField, 
				pValue := 0, cbValue := 0,
				bCRLF := ( nColumn = MAX_CSV_COLUMNS ) );
IF fbWriter.bOk THEN
	fbWriter.eCmd := eEnumCmd_Next;
ELSE
	step := 100;
RETURN;
END_IF
IF RIGHT( sCSVLine, 2 ) = '$R$L' THEN
	sCSVLine := REPLACE( sCSVLine, '$L', 2, LEN( sCSVLine ) - 1 );
END_IF
END_FOR
	nRow := nRow + 1;
	step := 4;
END_IF
END_IF
	4:	
	fbFilePuts( bExecute := FALSE );
	fbFilePuts( sNetId := sNetId, hFile := hFile, sLine := sCSVLine, bExecute := TRUE );
	step := 5;
	5:
	fbFilePuts( bExecute := FALSE, bError => bError, nErrID => nErrID );
IF NOT fbFilePuts.bBusy THEN
IF NOT fbFilePuts.bError THEN
	step := 3;
ELSE
	step := 100;
END_IF
END_IF
	10:	
	fbFileClose( bExecute := FALSE );
	fbFileClose( sNetId := sNetId, hFile := hFile, bExecute := TRUE );
	step := 11;
	11:
	fbFileClose( bExecute := FALSE, bError => bError, nErrID => nErrID );
IF ( NOT fbFileClose.bBusy ) THEN
	hFile := 0;
	step := 100;
END_IF
	100: 
IF ( hFile <> 0 ) THEN
	step := 10; 
ELSE
	bBusy := FALSE;
	step := 0;
	bWrite:=TRUE;//循环写入
END_IF
END_CASE

END_PROGRAM

// ---- POUs/报警/FB_SetAlarm.TcPOU
FUNCTION_BLOCK FB_SetAlarm(*设置报警功能块,每个报警调用一次*)
(*===========================================
by Swen 陈颂文
GuangZhou
2009-08-26

20171122转化成TC3   Swen

===========================================*)
VAR_INPUT
    InUse:                         	BOOL;(*是否使用*)
	EventId:						INT;(*报警号*)
	EventMessage:                  	STRING;(*报警信息*)
	EventActive:					BOOL;(*触发信号*)
   	FilterInUse:                  	BOOL:=FALSE;(* 是否使用滤波器*)(*对触发信号进行滤波，就是触发信号超过多少时间后才报警*)
   	FilterTime:                    	TIME;(*滤波时间*)
	QuitRequired:					BOOL;(*是否自动复位: true=复位信号为1时复位报警信号;false=触发信号为0时复位报警信号*)
	QuitEvent:					 	BOOL;(*复位信号*)
	EventClass:						Alm_EventClass;(*报警等级*)
	ToTheLogFile:					BOOL;(*是否记录到历史记录文件*)
   	ToTheHistory:                 	BOOL;(*是否记录到报警历史记录*)
	(* event actions	*)
	AlarmlampOn:				BOOL;(*是否需要报警灯亮*)
	AutoRunOff:					BOOL;(*退出自动循环*)
	AlarmAction1:				BOOL;(*用户定义报警动作*)(*例如定义为黄灯亮,则该报警号有触发时,主报警程序的该输出信号为1*)
	AlarmAction2:				BOOL;(*用户定义报警动作*)
	AlarmAction3:				BOOL;(*用户定义报警动作*)
	AlarmAction4:				BOOL;(*用户定义报警动作*)
	AlarmAction5:				BOOL;(*用户定义报警动作*)
	AlarmAction6:				BOOL;(*用户定义报警动作*)
	AlarmAction7:				BOOL;(*用户定义报警动作*)
	AlarmAction8:				BOOL;(*用户定义报警动作*)	
	D1:							DINT;//20171122 swen新增加
	D2:							DINT;//20171122 swen新增加
	S1:							STRING(80);//20171122 swen新增加
END_VAR
VAR_OUTPUT
	EventAlive:					BOOL;(*当前报警正在执行*)
  	ShowlampOn:            		BOOL;(*当前报警灯亮*)
END_VAR
VAR
 	F_Trig_QuitEvent:          	F_TRIG;
	n:                        	INT;
	R_TRIG_GetTime:          	R_TRIG;
  	TON_Filter:               	TON;
	sTemp: 						STRING;
	fbFormatStringDateTime: 	FB_FormatString;
	swFormatWstring: 			SW_FormatWstring;
	sDateTimeString: 			STRING(255);
	wEventMessage: 				WSTRING;
END_VAR

IF EventId> cnAlarmLast
OR EventId< cnAlarmFirst THEN
	RETURN;
END_IF

(*--------------------------------------------------警报数组---------------------------------------------------*)
       (*Reset Alarm*)
	   F_Trig_QuitEvent(CLK:=QuitEvent);
       	IF (QuitRequired AND  F_Trig_QuitEvent.Q)
      	OR NOT QuitRequired AND NOT EventActive
     	OR NOT InUse THEN
              	EventAlive:=FALSE;
            	ShowlampOn:=FALSE;
				AlarmActionArray[EventId].AutoRunOff	:=FALSE;(*退出自动循环*)
             	AlarmActionArray[EventId].AlarmAction1:=FALSE;
             	AlarmActionArray[EventId].AlarmAction2:=FALSE;
            	AlarmActionArray[EventId].AlarmAction3:=FALSE;
             	AlarmActionArray[EventId].AlarmAction4:=FALSE;
             	AlarmActionArray[EventId].AlarmAction5:=FALSE;
             	AlarmActionArray[EventId].AlarmAction6:=FALSE;
            	AlarmActionArray[EventId].AlarmAction7:=FALSE;
            	AlarmActionArray[EventId].AlarmAction8:=FALSE;
				AlarmActionArray[EventId].InUse:=InUse;
				AlarmActionArray[EventId].EventAlive:=EventAlive;
				AlarmActionArray[EventId].ShowlampOn:=ShowlampOn;
				AlarmActionArray[EventId].EventActive:=EventActive;
				AlarmActionArray[EventId].EventClass:=EventClass;
				AlarmActionArray[EventId].EventId:=EventId;
				AlarmActionArray[EventId].QuitEvent:=QuitEvent;
				AlarmActionArray[EventId].QuitRequired:=QuitRequired;
				AlarmActionArray[EventId].ShowlampOn:=ShowlampOn;
       	END_IF
(*-----------------------------------------------当前激活警报数组-------------------------------------------------*)	
       (*SetAlarm*)
	 	TON_Filter(IN:=FilterInUse AND EventActive , PT:=FilterTime );
		R_TRIG_GetTime(CLK:=(NOT FilterInUse AND EventActive) OR (FilterInUse AND TON_Filter.Q)AND InUse );  
		IF R_TRIG_GetTime.Q THEN
      		AlarmActionArray[EventId].EventTime:=SYSTEMTIME_TO_DT(tActSystemTime);
		END_IF
       	IF ((NOT FilterInUse AND EventActive) OR (FilterInUse AND TON_Filter.Q)) 
		AND InUse THEN
              EventAlive:=TRUE;
              ShowlampOn:=AlarmlampOn;
              AlarmActionArray[EventId].AutoRunOff:=AutoRunOff;
              AlarmActionArray[EventId].AlarmAction1:=AlarmAction1;
              AlarmActionArray[EventId].AlarmAction2:=AlarmAction2;
              AlarmActionArray[EventId].AlarmAction3:=AlarmAction3;
              AlarmActionArray[EventId].AlarmAction4:=AlarmAction4;
              AlarmActionArray[EventId].AlarmAction5:=AlarmAction5;
              AlarmActionArray[EventId].AlarmAction6:=AlarmAction6;
              AlarmActionArray[EventId].AlarmAction7:=AlarmAction7;
              AlarmActionArray[EventId].AlarmAction8:=AlarmAction8;
			  (*I/O*)
			 AlarmActionArray[EventId].InUse:=InUse;
			 AlarmActionArray[EventId].EventAlive:=EventAlive;
			 AlarmActionArray[EventId].ShowlampOn:=ShowlampOn;
			 AlarmActionArray[EventId].EventActive:=EventActive;
			 AlarmActionArray[EventId].EventClass:=EventClass;
			 AlarmActionArray[EventId].EventId:=EventId;
			 IF R_TRIG_GetTime.Q THEN
				 fbFormatStringDateTime(
					sFormat:= 	'%D-%D-%D-%D:%D:%D',
					arg1:= 		F_WORD(tActSystemTime.wYear),
					arg2:= 		F_WORD(tActSystemTime.wMonth),
					arg3:= 		F_WORD(tActSystemTime.wDay),
					arg4:= 		F_WORD(tActSystemTime.wHour),
					arg5:= 		F_WORD(tActSystemTime.wMinute),
					arg6:= 		F_WORD(tActSystemTime.wSecond),
					sOut=> 		sDateTimeString
					);
				IF CurrentLanguage='English' THEN
					wEventMessage:=STRING_TO_WSTRING(AlarmActionArray[EventId].AlarmMsg.EN);
				ELSE
					wEventMessage:=AlarmActionArray[EventId].AlarmMsg.CN;
				END_IF
				
				swFormatWstring(
					WstringIn:= 	wEventMessage, 
					D1:= 			D1, 
					D2:= 			D2, 
					S1:= 			S1, 
					WstringOUT=> 	wEventMessage
					);
	
				wEventMessage:=	WCONCAT(WCONCAT(WCONCAT(
										"ID",
										INT_TO_WSTRING(EventId)),
										","),
										wEventMessage);
		
				AlarmActionArray[EventId].EventMessage := WCONCAT(WCONCAT(
															STRING_TO_WSTRING(sDateTimeString),
															"-"),
															wEventMessage);	
			END_IF
			
			AlarmActionArray[EventId].QuitEvent:=QuitEvent;
			AlarmActionArray[EventId].QuitRequired:=QuitRequired;
			AlarmActionArray[EventId].ShowlampOn:=ShowlampOn;
       END_IF
	   
(*---------------------------------------------------历史警报数组----------------------------------------------------*)
IF ToTheHistory  
AND R_TRIG_GetTime.Q THEN
        Alm_HistoryAlarmNum:=Alm_HistoryAlarmNum+1;
        IF Alm_HistoryAlarmNum>=cnAlmHistoryLast THEN
               Alm_HistoryAlarmNum:=cnAlmHistoryLast;
        END_IF
        IF Alm_HistoryAlarmNum>=cnAlmHistoryFirst+1 THEN
             FOR n:=Alm_HistoryAlarmNum TO cnAlmHistoryFirst+1 BY -1 DO
                  AlarmHistoryArray[n]:=AlarmHistoryArray[n-1];
             END_FOR
        END_IF
 	AlarmHistoryArray[1].EventId:=EventId;
	AlarmHistoryArray[1].EventTime:=AlarmActionArray[EventId].EventTime;
  	AlarmHistoryArray[1].EventMessage:=AlarmActionArray[EventId].EventMessage;
END_IF
IF ToTheLogFile
AND R_TRIG_GetTime.Q THEN
	wstring_to_utf8(ADR(sTemp),ADR(wEventMessage),SIZEOF(sTemp));
	gsWriteToLog:=concat(gsWriteToLog,sTemp);
END_IF

END_FUNCTION_BLOCK

// ---- POUs/报警/SW_FormatWstring.TcPOU
FUNCTION_BLOCK SW_FormatWstring
//格式化字符串
//SwenChen
//20171123
VAR_INPUT
	WstringIn:			WSTRING;
	D1:					DINT;
	D2:					DINT;
	S1:					STRING;
END_VAR
VAR_OUTPUT
	WstringOUT:			WSTRING;
END_VAR
VAR
	Var1: 				INT;
END_VAR


Var1:=WFIND(WstringIn,"%D");
IF Var1<>0 THEN
	WstringOUT := WREPLACE(WstringIn,DINT_TO_WSTRING(D1),2,Var1);

	Var1:=WFIND(WstringOUT,"%D");
	IF Var1<>0 THEN
		WstringOUT := WREPLACE(WstringOUT,DINT_TO_WSTRING(D2),2,Var1);
	END_IF
ELSE
	WstringOUT:=WstringIN;
END_IF

Var1:=WFIND(WstringOUT,"%S");
IF Var1<>0 THEN
	WstringOUT := WREPLACE(WstringOUT,STRING_TO_WSTRING(S1),2,Var1);
END_IF

END_FUNCTION_BLOCK

// ---- DUTs/文件配方/FB_FileOperate.TcPOU
FUNCTION_BLOCK FB_FileOperate
VAR_INPUT
END_VAR
VAR_OUTPUT
END_VAR
VAR
	Step: USINT := 0;								(* Step of the FB *)
	Index: USINT := 0;								(* Index for variable to be loaded or saved*)
	FB_XmlSrvReadByName: FB_XmlSrvReadByName;		(* Read the variable by name in the xml file*)
	FB_FormatString: FB_FormatString;				(* Convert the name to configed format string *)
	FB_XmlSrvWriteByName: FB_XmlSrvWriteByName;		(* Save the variable value by name in the XML file *)
END_VAR
VAR_IN_OUT
	CMD: File_com_typ;		(* Command of the file operatation *)
END_VAR
VAR CONSTANT
	COMMAND: USINT := 0;		(* *)
	FILE_SAVE: USINT := 10;
	FILE_SAVE_PROCESS: USINT := 11;

	FILE_LOAD: USINT := 20;
	FILE_LOAD_PROCESS: USINT := 21;

	FILE_DELETE: USINT := 90;

END_VAR

CASE Step OF
	COMMAND:
		CMD.bBusy := FALSE;
		IF CMD.File_load THEN
			Index 	:= 0;
			IF CMD.Var_Name[Index] <> '' THEN
				Step 	:= FILE_LOAD;
				CMD.bBusy := TRUE;
				CMD.File_load := 0;
			ELSE
			 	CMD.ErrorID := 10001;		(*No variable name config*)
			END_IF
		END_IF

		IF CMD.File_save THEN
			Index 	:= 0;
			IF CMD.Var_Name[Index] <> '' THEN
				Step := FILE_SAVE;
				CMD.bBusy := TRUE;
				CMD.File_save := 0;
			ELSE
			 	CMD.ErrorID := 10001;		(*No variable name config*)
			END_IF
		END_IF

	FILE_LOAD:
		(* Set the name of the Global variables *)
		FB_FormatString(sFormat:= '.%s', arg1:= F_STRING(CMD.Var_Name[Index]));
		FB_XmlSrvReadByName.sSymName := FB_FormatString.sOut;
		(* Set the format name of the Global variables in the xml file*)
		FB_FormatString(sFormat:= '/dataentry/%s', arg1:= F_STRING(CMD.Var_Name[Index]));
		FB_XmlSrvReadByName.sXPath := FB_FormatString.sOut;
		(* Set the file path name *)
		FB_FormatString(sFormat:= '%s%s', arg1:= F_STRING(CMD.Device), arg2 := F_STRING(CMD.FileName_active));
		FB_XmlSrvReadByName.sFilePath := FB_FormatString.sOut;

		FB_XmlSrvReadByName(
			nMode:= XMLSRV_ADDMISSING,
			bExecute:= TRUE,
		 );
		Index := Index + 1;
		Step := FILE_LOAD_PROCESS;


	FILE_LOAD_PROCESS:
		FB_XmlSrvReadByName(bExecute:= FALSE );

		IF NOT FB_XmlSrvReadByName.bBusy THEN
			IF CMD.Var_Name[Index] <> '' THEN
				Step 	:= FILE_LOAD;
			ELSE
			 	Step := COMMAND;

			END_IF

		END_IF
		CMD.ErrorID := FB_XmlSrvReadByName.nErrId;

	FILE_SAVE:
		(* Set the name of the Global variables *)
		FB_FormatString(sFormat:= '.%s', arg1:= F_STRING(CMD.Var_Name[Index]));
		FB_XmlSrvWriteByName.sSymName := FB_FormatString.sOut;
		(* Set the format name of the Global variables in the xml file*)
		FB_FormatString(sFormat:= '/dataentry/%s', arg1:= F_STRING(CMD.Var_Name[Index]));
		FB_XmlSrvWriteByName.sXPath := FB_FormatString.sOut;
		(* Set the file path name *)
		FB_FormatString(sFormat:= '%s%s', arg1:= F_STRING(CMD.Device), arg2 := F_STRING(CMD.FileName_save));
		FB_XmlSrvWriteByName.sFilePath := FB_FormatString.sOut;

		FB_XmlSrvWriteByName(
			nMode:= XMLSRV_ADDMISSING,
			bExecute:= TRUE,
		 );
		Index := Index + 1;
		Step := FILE_SAVE_PROCESS;

	FILE_SAVE_PROCESS:
		FB_XmlSrvWriteByName(bExecute:= FALSE );

		IF NOT FB_XmlSrvWriteByName.bBusy THEN
			IF CMD.Var_Name[Index] <> '' THEN
				Step 	:= FILE_SAVE;
			ELSE
			 	Step := COMMAND;

			END_IF

		END_IF
		CMD.ErrorID := FB_XmlSrvWriteByName.nErrId;
END_CASE

END_FUNCTION_BLOCK

// ---- DUTs/文件配方/Swen_Products/FB_FileCopy_lib.TcPOU
FUNCTION_BLOCK FB_FileCopy_lib
VAR_INPUT
	srcNetId		: T_AmsNetId;	(* TwinCAT network address of the source file *)
	srcFileName	: T_MaxString;	(* source file path and name *)
	destNetId		: T_AmsNetId;	(* TwinCAT network address of the destination file *)
	destFileName	: T_MaxString;  	(* destination file path and name *)
	bExecute		: BOOL;		(* rising edge starts fb execution *)
	tAdsTimeOut	: TIME;		(* ads timeout *)
END_VAR
VAR_OUTPUT
	bBusy		:BOOL;
	bError		:BOOL;
	nErrId		:UDINT;
END_VAR
VAR
	fbFileOpen	:FB_FileOpen;
	fbFileClose	:FB_FileClose;
	fbFileRead	:FB_FileRead;
	fbFileWrite	:FB_FileWrite;

	hSrcFile		:UINT	:= 0;(* file handle of the source file *)
	hDestFile		:UINT	:= 0;(* file handle of the destination file *)

	Step		:DWORD;
	RisingEdge	:R_TRIG;

	buffRead		:ARRAY[1..100] OF BYTE;(* buffer *)
	cbReadLength	:UDINT:=0;
END_VAR

RisingEdge(CLK:=bExecute);
IF RisingEdge.Q THEN
	IF NOT bBusy THEN
		bBusy := TRUE;
		bError:= FALSE;
		nErrId:=0;
		Step := 1;
		cbReadLength:=0;
		hSrcFile:=0;
		hDestFile:=0;
	END_IF
END_IF


CASE Step OF
	0:(* do nothing *)
	;

	1:(* open source file *)
	fbFileOpen(  bExecute := FALSE  );
	fbFileOpen(	sNetId := srcNetId,
		sPathName := srcFileName,
		nMode := FOPEN_MODEREAD OR FOPEN_MODEBINARY,
		ePath := PATH_GENERIC,
		tTimeout := tAdsTimeout,
		bExecute := TRUE );
		Step := Step + 1;

	2:
	fbFileOpen( bExecute := FALSE );
	IF ( NOT fbFileOpen.bBusy ) THEN
		IF ( fbFileOpen.bError ) THEN
			nErrId := fbFileOpen.nErrId;
			bError := TRUE;
			Step := 50;
		ELSE
			hSrcFile := fbFileOpen.hFile;
			Step := Step + 1;
		END_IF
	END_IF

	3:(* open destination file *)
	fbFileOpen(  bExecute := FALSE  );
	fbFileOpen( 	sNetId := destNetId,
			sPathName := destFileName,
			nMode := FOPEN_MODEWRITE OR FOPEN_MODEBINARY,
			ePath := PATH_GENERIC,
			tTimeout := tAdsTimeout,
			bExecute := TRUE );
	Step := Step+1;

	4:
	fbFileOpen(  bExecute := FALSE  );
	IF ( NOT fbFileOpen.bBusy ) THEN
		IF ( fbFileOpen.bError ) THEN
			nErrId := fbFileOpen.nErrId;
			bError := TRUE;
			Step := 50;
		ELSE
			hDestFile := fbFileOpen.hFile;
			Step := Step + 1;
		END_IF
	END_IF

	5:(*read data from source file*)
	cbReadLength := 0;
	fbFileRead( bExecute:= FALSE );
	fbFileRead( 	sNetId:=SrcNetId,
			hFile:=hSrcFile,
			pReadBuff:= ADR(buffRead),
			cbReadLen:= SIZEOF(buffRead),
			bExecute:=TRUE,
			tTimeout:=tAdsTimeOut );
	Step := Step + 1;

	6:
	fbFileRead( bExecute:= FALSE );
	IF ( NOT fbFileRead.bBusy ) THEN
		IF ( fbFileRead.bError ) THEN
			nErrId := fbFileRead.nErrId;
			bError := TRUE;
			Step := 50;
		ELSE
			cbReadLength := fbFileRead.cbRead;
			Step := Step + 1;
		END_IF
	END_IF

	7:(*write data to destination file*)
	fbFileWrite( bExecute := FALSE );
	fbFileWrite(	sNetId:=DestNetId,
			hFile:=hDestFile,
			pWriteBuff:= ADR(buffRead),
			cbWriteLen:= cbReadLength,
			bExecute:=TRUE,
			tTimeout:=tAdsTimeOut );
	Step := Step + 1;

	8:
	fbFileWrite( bExecute := FALSE );
	IF ( NOT fbFileWrite.bBusy ) THEN
		IF ( fbFileWrite.bError ) THEN
			nErrId := fbFileWrite.nErrId;
			bError := TRUE;
			Step := 50;
		ELSE
			IF fbFileRead.bEOF THEN (*Check if the EOF flag ist set *)
				Step := 50;(*cleanup: close the destination and source files *)
			ELSE
				Step := 5; (* repeat reading *)
			END_IF
		END_IF
	END_IF

	30:(* close the destination file *)
	fbFileClose( bExecute := FALSE );
	fbFileClose( 	sNetId:=destNetId,
			hFile:=hDestFile,
			bExecute:=TRUE,
			tTimeout:=tAdsTimeOut );
	Step := Step + 1;

	31:
	fbFileClose( bExecute := FALSE );
	IF ( NOT fbFileClose.bBusy ) THEN
		IF ( fbFileClose.bError ) THEN
			nErrId := fbFileClose.nErrId;
			bError := TRUE;
		END_IF
		Step := 50;
		hDestFile := 0;
	END_IF

	40: (* close source file *)
	fbFileClose( bExecute := FALSE );
	fbFileClose( 	sNetId:=srcNetId,
			hFile:=hSrcFile,
			bExecute:=TRUE,
			tTimeout:=tAdsTimeOut );
	Step := Step + 1;

	41:
	fbFileClose( bExecute := FALSE );
	IF ( NOT fbFileClose.bBusy ) THEN
		IF ( fbFileClose.bError ) THEN
			nErrId := fbFileClose.nErrId;
			bError := TRUE;
		END_IF
		Step := 50;
		hSrcFile := 0;
	END_IF

	50: (*error or ready => cleanup*)
	IF ( hDestFile <> 0 ) THEN
		Step := 30; (* close the destination file*)
	ELSIF (hSrcFile <> 0 ) THEN
		Step := 40; (* close the source file *)
	ELSE
		Step := 0;	(* ready *)
		bBusy := FALSE;
	END_IF

END_CASE

END_FUNCTION_BLOCK
